# B&R Automation Studio project dbserv_0640 (part 5)

#### dbserv.c
```c
#ifdef _DEFAULT_INCLUDES
	#include <AsDefault.h>
#endif

/******************************************************************************
*    COPYRIGHT    BERNECKER + RAINER Industrie-Elektronik Ges.m.b.H           *
*******************************************************************************
*  Projekt:  DbServ
*  Teil:     Prozessabbild-Aufbau
*  Datei:    dbserv.c
*  Typ:      GNU-C (32 Bit)
*------------------------------------------------------------------------------
*  Revision: 01.03
*  Datum:    26-07-2004
*  Autor:    Martin Kurtz / MKrz
*------------------------------------------------------------------------------
*  Funktion: Task-Source-Datei.
*------------------------------------------------------------------------------
*  Rev.  | Datum    | Name | Kommentar
*  ------+----------+------+---------------------------------------------------
*  01.03 | 26-07-04 | MKrz | Nichtangabe von Item.Name für nicht verwendete Fubinstanzen
*        |          |      | führt zu keinen Logbucheinträgen;
*  01.02 | 15-07-04 | MKrz | Fehlerbeseitigung bei Logbuch-Fehlereintrag;
*  01.01 | 06-07-04 | MKrz | Fehlerbeseitigung Eventblockverwaltung;
*        |          |      | Parserfunktion für Timeout, Port, Client.Anz, App.Anz
*  01.00 | 04-08-03 | MKrz | Datei-Erstellung
*  02.00 | 10-07-26 | BIE  | strnicmp gegen strncasecmp ersetzt
*        |          |      |
******************************************************************************/

/***********************************************************************/
/* Headerfiles einbinden                                               */
/***********************************************************************/
#include <bur\plc.h>		/* RPS-spezifische Typendeklarationen */
#include <sys_lib.h>		/* System-Library */

#include <dataobj.h>
#include <fileio.h>
#include <brsystem.h>

#include <string.h>			/* String-Library */
#include <stdlib.h>			/* String-Library */

#include "platform.h"		/* CPU-Plattform */

#include "bksys.h"			/* Burklimat-Library */

#include "parser.h"			/* Parser-Library */
#include "dbserv.h"			/* BkTcp-Library */

#include <dbslib.h>

//unsigned short itoa(signed long value, unsigned long pString);

/***********************************************************************/
/* Variablendeklaration                                                */
/***********************************************************************/

/**** globale Variablen ************************************************/

/**** lokale Variablen *************************************************/

/* Anzahl Fehlerzaehler fuer ErrStatistics */
/*#define ERRCNTANZ				300*/

/* Struktur fuer Fehler-Statistik */
/*typedef struct {
	unsigned short	LastWarn;
	unsigned short	LastErr;
	unsigned short	Init;
	Timestamp_Typ	LastInit;
	unsigned short	ErrCount[ERRCNTANZ];
} Stats_Typ;*/

_LOCAL_RETAIN Stats_Typ		SYS_Statistic	;

_LOCAL_RETAIN	unsigned short	ParserState	;

_LOCAL_RETAIN	BIT				DbsTypeChanged, DbsPointChanged	;
		void  			*pDA_Data;
_LOCAL_RETAIN	UDINT			SizeDA_Data	;

_LOCAL	DatObjInfo_typ		iDatObjInfo;
_LOCAL	DatObjDelete_typ	iDatObjDelete;
_LOCAL	DatObjCreate_typ	iDatObjCreate;

_LOCAL_RETAIN	unsigned short	CountLines	;
_LOCAL_RETAIN	signed short	State_find_StationTypPoint, State_find_Section, State_find_Data	;
		short			StateGetDpInfo;

		unsigned char	*pParser, *pParserLine, *pParserErr;
		unsigned short	SectionType;
		unsigned char	*pDataArg1, *pDataArg2, *pDataArg3, *pTempStation, *pTempSection, *pTempPoint, *pTempData, *pDbsTypeFileBufferSize, *pDbsTypeFileBufferMode;
		unsigned short	SizeArg1, SizeArg2, SizeArg3 ;

_LOCAL	unsigned short	PortNumber, TimeoutValue;
_LOCAL	long			BufEvents, BufType;

		unsigned char	flagDbsUnit, flagDbsType, flagDbsPoint, flagDbsFub, flag, flagDbsExistPoints, flagDbsNotExistPoints, flagDbsFubInstance;
_LOCAL_RETAIN	unsigned short	maxDbsUnit, maxUsedUnit, DbsUnit, DbsType, maxDbsType, maxUsedType, DbsPoint, DbsItem	;
_LOCAL	unsigned char	DbsMemTypeData, DbsMemTypeEvent;
_LOCAL_RETAIN	unsigned long	memSize, SmemSize, StmpSize	;
		unsigned short	StateTMP_alloc;

_LOCAL_RETAIN	unsigned short	countStationTypPoint, countSection, countItem, countTimeItem	;
_LOCAL	unsigned short	countDefinedType, countDefinedPoint, countDefinedItem, countPortData, countTimeoutData, countEventData, countTypeData, countUnitData, countPointData	;
_LOCAL	unsigned short	countFub, countData, countExistPoints, countNotExistPoints, countNotDefinedItems, countInvalidExistItems, countNotExistItems, countLogMessages, countFubInstance	;
_LOCAL_RETAIN	unsigned short	countEventInstance, countWriteInstance	;

_LOCAL	unsigned short	SizeNameType, SizeNamePoint, SizeNameItem, sizeType, lenItem	;
_LOCAL_RETAIN	unsigned char	sItem, idTypeItem	;

		char			logBuffer[128];
		unsigned short	sMsgMaxLen;
_LOCAL_RETAIN	short			SwVersion	;

		unsigned short	i, j;
		unsigned char	DtIdx;
		unsigned short	DpIdx;

_LOCAL_RETAIN	unsigned char	go	;
_LOCAL_RETAIN	short			AnzWaitCycleDbs	;
		unsigned char	ErrStatisticsYField[EC_MAX / 8 + 1];

_LOCAL	TYPE_DESC		*pTypeDesc, *pWorkTypeDesc, *pInfoTypeDesc;
_LOCAL	ITEM_DESC		*pItemDesc, *pWorkItemDesc, *pInfoItemDesc;
_LOCAL	POINT_DESC		*pPointDesc, *pWorkPointDesc, *pInfoPointDesc;
_LOCAL	FUB_DESC		*pFubInstanceDesc;
_LOCAL_RETAIN	unsigned short	infoType, infoPoint	;
_LOCAL_RETAIN	unsigned char	*pTypeName, *pWorkTypeName, *pPointName, *pWorkPointName, *pWorkItemName, InfoTypeName[16], PointName[64]	;
		unsigned short	lenTypeName, lenPointName;
		unsigned long	len;

_LOCAL	ACCESS_SERVER		*idBrServer,	*pAccessServer;
		ACCESS_UNIT			*pAccessUnit;
		ACCESS_TYPE			*pAccessType,	*pAccessTypeWork;
		ACCESS_POINT		*pAccessPoint,	*pAccessPointWork;
		ACCESS_DATA			*pAccessData,	*pAccessDataWork;
		ACCESS_FUB_INSTANCE	*pAccessFubInstance;

		ACCESS_EVENT_PIPE	*pEventPipe;
		EVENT_PIPE_INSTANCE	*pEventPipeInstance;
		EVENT_PIPE_HEADER	*pEventPipeHeader;
		ACCESS_WRITE_PIPE	*pWritePipe;
		WRITE_PIPE_HEADER	*pWritePipeHeader;

_LOCAL_RETAIN	UINT			stateFubInstance	;
_LOCAL	UDINT			pFubInstance, lenFubInstance	;

/*_LOCAL	FUB_REF			x;*/

_LOCAL_RETAIN	USINT		bValue	;
_LOCAL_RETAIN	RTCtime_typ	RTCTime	;

_LOCAL	FileCreate_typ	iFileCreate;
_LOCAL	DevMemInfo_typ	iDevMemInfo;
_LOCAL	BOOL	filetest;
_LOCAL	USINT	buffer1[32], buffer2[32];

_LOCAL	SysInfo_typ		iSysInfo;

/***********************************************************************/
/* Initialisierungs-Unterprogramm                                      */
/***********************************************************************/

void _INIT init(void)
{
	idBrServer = NULL;
	SwVersion = BK_VERSION_NR;

	SYS_Statistic = SYS_Statistic;

	PortNumber = cTCP_DEFAULT_PORT;
	TimeoutValue = cTCP_DEFAULT_TIMEOUT;

	BufEvents = 0;
	BufType = 0;

	ParserState = cCD_PARSER_STATE_DEF_TCP;
	memset(ErrStatisticsYField, 0, sizeof(ErrStatisticsYField));

	AnzWaitCycleDbs = 0;

	countEventInstance = 8;
	countWriteInstance = 4;

	DbsTypeChanged = TRUE;
	DbsPointChanged = TRUE;

	go = TRUE;
}

/***********************************************************************/
/* zyklisches Hauptprogramm                                            */
/***********************************************************************/
void _CYCLIC cyclic(void)
{
	if (filetest == TRUE) {
		strcpy(buffer1, "Test");
		ultoa(i, buffer2);
		strcat(buffer1, buffer2);

		iFileCreate.enable = 1;
		iFileCreate.pDevice = (unsigned long)"CompactFlash";
		iFileCreate.pFile = (unsigned long)buffer1;
		FileCreate(&iFileCreate);
		if (iFileCreate.status == 0) {
			filetest = FALSE;
			i++;
		}
		else if (iFileCreate.status != 65535) {
			filetest = FALSE;
			i++;
		}
	}

	/* ----------------- */
	/* Start-Verzögerung */
	/* ----------------- */
	if (AnzWaitCycleDbs < ANZ_WAIT_CYCLE_TCP) {
		AnzWaitCycleDbs++;
		return;
	}

	/* ------------- */
	/* Parser - Lauf */
	/* ------------- */
	if (go == TRUE) {

		/* --- */
		/* DFA */
		/* --- */
		/*while (ParserState < cCD_PARSER_STATE_READY) {*/

			/* ------------- */
			/* DFA - Zustand */
			/* ------------- */
			switch (ParserState) {

				/* ============================= */
				/* DFA-Zustand: Tcp-Definitionen */
				/* ============================= */
				case cCD_PARSER_STATE_DEF_TCP:

					iDatObjInfo.enable = TRUE;
					iDatObjInfo.pName = (UDINT)cKW_DBS_DM_DP_LIST;
					DatObjInfo(&iDatObjInfo);
					if (iDatObjInfo.status == 0) {
						pDA_Data = (unsigned char*)iDatObjInfo.pDatObjMem;
						SizeDA_Data = iDatObjInfo.len;

						/* go */

						/* Datenmodul von Anfang an Parsen ... */
						CountLines = 0;
						pParser = (unsigned char*)pDA_Data;

						/* Zähler rücksetzen */
						countPortData = 0;
						countTimeoutData = 0;
						countStationTypPoint = 0;

						/* Parser-Status loeschen */
						State_find_StationTypPoint = 0;
						State_find_Section = 0;
						State_find_Data = 0;

						/* ------ */
						/* Parsen */
						/* ------ */
						while (pParser < (unsigned char*)pDA_Data + SizeDA_Data) {

							/* Suche nach Stations/Typ/Punkt-Beschreibung */
							State_find_StationTypPoint = find_StationTypPoint(pDA_Data, pParser, pDA_Data + SizeDA_Data,
																				&pParser, &pParserLine, &pParserErr, &CountLines,
																				&pDataArg1, &SizeArg1,
																				&pDataArg2, &SizeArg2,
																				&SectionType);
							/* keine Daten oder Fehler aufgetreten ? */
							if (State_find_StationTypPoint < 0) {
								break;
							}
							else {
								countStationTypPoint++;
							}

							/* Pointer auf Station/Typ/Punkt */
							switch (SectionType) {

								/* ------------------ */
								/* Stations-Abschnitt */
								/* ------------------ */
								case cCD_STATION:
									countSection = 0;
									do {
										State_find_Section = find_Section(pDA_Data, pParser, pDA_Data + SizeDA_Data,
																			&pParser, &pParserLine, &pParserErr, &CountLines,
																			&pDataArg1, &SizeArg1,
																			&pDataArg2, &SizeArg2,
																			cKW_TCP_SECTION);
										/* keine Daten oder Fehler aufgetreten ? */
										if (State_find_Section < 0) {
											break;
										}
										else {
											countSection++;
										}

										/* Pointer auf Anfang der Sektion stellen */
										if (pDataArg2 != NULL) {
											pParser = pDataArg2;
										}
										else {
											continue;
										}

										/* alle Daten der Sektion bearbeiten */
										countData = 0;
										do {
											/* Daten der Sektion anfordern */
											State_find_Data = find_Data(pDA_Data, pParser, pDA_Data + SizeDA_Data,
																		  &pParser, &pParserLine, &pParserErr, NULL,
																		  &pDataArg1, &SizeArg1,
																		  &pDataArg2, &SizeArg2,
																		  &pDataArg3, &SizeArg3);
											/* keine Daten oder Fehler aufgetreten ? */
											if (State_find_Data < -1) {
												break;
											}
											else if (State_find_Data == -1) {
												if (pParser < (unsigned char*)pDA_Data + SizeDA_Data) {
													pParser++;
													State_find_Data = TRUE;
													continue;
												}
												else {
													break;
												}
											}
											else {
												/* Port-Bezeichner */
												if (strlen(cKW_TCP_PORT) == SizeArg1 && strncasecmp(pDataArg1, cKW_TCP_PORT, SizeArg1) == 0 &&
													strlen(cKW_TCP_PORT_NUMBER) == SizeArg2 && strncasecmp(pDataArg2, cKW_TCP_PORT_NUMBER, SizeArg2) == 0 &&
													pDataArg3 != NULL && SizeArg3 != 0 &&
													IsANumber(pDataArg3) == TRUE)
												{
													countPortData++;
													PortNumber = atoi(pDataArg3);
												}
												/* Timeout-Bezeichner */
												else if (strlen(cKW_TCP_TIMEOUT) == SizeArg1 && strncasecmp(pDataArg1, cKW_TCP_TIMEOUT, SizeArg1) == 0 &&
													strlen(cKW_TCP_TIMEOUT_NUMBER) == SizeArg2 && strncasecmp(pDataArg2, cKW_TCP_TIMEOUT_NUMBER, SizeArg2) == 0 &&
													pDataArg3 != NULL && SizeArg3 != 0 &&
													IsANumber(pDataArg3) == TRUE)
												{
													countTimeoutData++;
													TimeoutValue = atoi(pDataArg3);
												}
												/* unbekannte Zuweisung */
												else {
												}
											}
										} while (State_find_Data == TRUE);
									} while (State_find_Section == TRUE);
									break;
							} /* (SectionType) */
						} /* (pParser < (unsigned char*)pDA_Data + SizeDA_Data) */

						/* ---------------- */
						/* nächster Zustand */
						/* ---------------- */
						ParserState = cCD_PARSER_STATE_DEF_BUF;

					} /* (DA_DataOk == TRUE) */
					else {
						/* Fehler beim Datenmodul */
						ErrStatistics("dbserv", ERRLOG, EC_DA_NOT_FOUND + EC_DBS_BASE, CountLines, ERR_DBS_PRE, ET_DA_NOT_FOUND);
						ParserState = cCD_PARSER_STATE_ERROR;
					}
					break;

				/* ============================= */
				/* DFA-Zustand: Buf-Definitionen */
				/* ============================= */
				case cCD_PARSER_STATE_DEF_BUF:

					iDatObjInfo.enable = TRUE;
					iDatObjInfo.pName = (UDINT)cKW_DBS_DM_DP_LIST;
					DatObjInfo(&iDatObjInfo);
					if (iDatObjInfo.status == 0) {
						pDA_Data = (unsigned char*)iDatObjInfo.pDatObjMem;
						SizeDA_Data = iDatObjInfo.len;

						/* go */

						/* Datenmodul von Anfang an Parsen ... */
						CountLines = 0;
						pParser = (unsigned char*)pDA_Data;

						/* Zähler rücksetzen */
						countEventData = 0;
						countTypeData = 0;
						countStationTypPoint = 0;

						/* Parser-Status loeschen */
						State_find_StationTypPoint = 0;
						State_find_Section = 0;
						State_find_Data = 0;

						/* ------ */
						/* Parsen */
						/* ------ */
						while (pParser < (unsigned char*)pDA_Data + SizeDA_Data) {

							/* Suche nach Stations/Typ/Punkt-Beschreibung */
							State_find_StationTypPoint = find_StationTypPoint(pDA_Data, pParser, pDA_Data + SizeDA_Data,
																				&pParser, &pParserLine, &pParserErr, &CountLines,
																				&pDataArg1, &SizeArg1,
																				&pDataArg2, &SizeArg2,
																				&SectionType);
							/* keine Daten oder Fehler aufgetreten ? */
							if (State_find_StationTypPoint < 0) {
								break;
							}
							else {
								countStationTypPoint++;
							}

							/* Pointer auf Station/Typ/Punkt */
							switch (SectionType) {

								/* ------------------ */
								/* Stations-Abschnitt */
								/* ------------------ */
								case cCD_STATION:
									countSection = 0;
									do {
										State_find_Section = find_Section(pDA_Data, pParser, pDA_Data + SizeDA_Data,
																			&pParser, &pParserLine, &pParserErr, &CountLines,
																			&pDataArg1, &SizeArg1,
																			&pDataArg2, &SizeArg2,
																			cKW_BUF_SECTION);
										/* keine Daten oder Fehler aufgetreten ? */
										if (State_find_Section < 0) {
											break;
										}
										else {
											countSection++;
										}

										/* Pointer auf Anfang der Sektion stellen */
										if (pDataArg2 != NULL) {
											pParser = pDataArg2;
										}
										else {
											continue;
										}

										/* alle Daten der Sektion bearbeiten */
										countData = 0;
										do {
											/* Daten der Sektion anfordern */
											State_find_Data = find_Data(pDA_Data, pParser, pDA_Data + SizeDA_Data,
																		  &pParser, &pParserLine, &pParserErr, NULL,
																		  &pDataArg1, &SizeArg1,
																		  &pDataArg2, &SizeArg2,
																		  &pDataArg3, &SizeArg3);
											/* keine Daten oder Fehler aufgetreten ? */
											if (State_find_Data < -1) {
												break;
											}
											else if (State_find_Data == -1) {
												if (pParser < (unsigned char*)pDA_Data + SizeDA_Data) {
													pParser++;
													State_find_Data = TRUE;
													continue;
												}
												else {
													break;
												}
											}
											else {
												/* Events-Bezeichner */
												if (strlen(cKW_DBS_BUF_EVENTS) == SizeArg1 && strncasecmp(pDataArg1, cKW_DBS_BUF_EVENTS, SizeArg1) == 0 &&
													pDataArg2 == NULL &&
													pDataArg3 != NULL && SizeArg3 != 0 &&
													IsANumber(pDataArg3) == TRUE)
												{
													countEventData++;
													BufEvents = atoi(pDataArg3);
												}
												/* Typ-Bezeichner */
												else if (strlen(cKW_DBS_BUF_TYPE) == SizeArg2 && strncasecmp(pDataArg2, cKW_DBS_BUF_TYPE, SizeArg2) == 0 &&
													pDataArg2 == NULL &&
													pDataArg3 != NULL && SizeArg3 != 0 &&
													IsANumber(pDataArg3) == TRUE)
												{
													countTypeData++;
													BufType = atoi(pDataArg3);
												}
												/* unbekannte Zuweisung */
												else {
												}
											}
										} while (State_find_Data == TRUE);
									} while (State_find_Section == TRUE);
									break;
							} /* (SectionType) */
						} /* (pParser < (unsigned char*)pDA_Data + SizeDA_Data) */

						/* ---------------- */
						/* nächster Zustand */
						/* ---------------- */
						ParserState = cCD_PARSER_STATE_COUNT_TYPE;

					} /* (DA_DataOk == TRUE) */
					else {
						/* Fehler beim Datenmodul */
						ErrStatistics("dbserv", ERRLOG, EC_DA_NOT_FOUND + EC_DBS_BASE, CountLines, ERR_DBS_PRE, ET_DA_NOT_FOUND);
						ParserState = cCD_PARSER_STATE_ERROR;
					}
					break;

				/* ====================================== */
				/* DFA-Zustand: Zählen der DBS-Datentypen */
				/* ====================================== */
				case cCD_PARSER_STATE_COUNT_TYPE:

					idBrServer = NULL;

					iDatObjInfo.enable = TRUE;
					iDatObjInfo.pName = (UDINT)cKW_DBS_DM_TYP_LIST;
					DatObjInfo(&iDatObjInfo);
					if (iDatObjInfo.status == 0) {
						pDA_Data = (unsigned char*)iDatObjInfo.pDatObjMem;
						SizeDA_Data = iDatObjInfo.len;

						SmemSize = 0, StmpSize = 0;

						/* go */

						/* Datenmodul von Anfang an Parsen ... */
						CountLines = 0;
						pParser = (unsigned char*)pDA_Data;

						/* Zähler rücksetzen */
						countDefinedType = 0;
						countDefinedItem = 0;
						countPortData = 0;
						countTimeoutData = 0;
						countExistPoints = 0;
						countNotExistPoints = 0;
						countStationTypPoint = 0;
						countLogMessages = 0;

						SizeNameType = 0, SizeNameItem = 0;

						/* Parser-Status loeschen */
						State_find_StationTypPoint = 0;
						State_find_Section = 0;
						State_find_Data = 0;

						/* ------ */
						/* Parsen */
						/* ------ */
						while (pParser < (unsigned char*)pDA_Data + SizeDA_Data) {

							/* Suche nach Stations/Typ/Punkt-Beschreibung */
							State_find_StationTypPoint = find_StationTypPoint(pDA_Data, pParser, pDA_Data + SizeDA_Data,
																				&pParser, &pParserLine, &pParserErr, &CountLines,
																				&pDataArg1, &SizeArg1,
																				&pDataArg2, &SizeArg2,
																				&SectionType);
							/* keine Daten oder Fehler aufgetreten ? */
							if (State_find_StationTypPoint < 0) {
								break;
							}
							else {
								countStationTypPoint++;
							}

							/* Pointer auf Station/Typ/Punkt */
							switch (SectionType) {

								/* ------------- */
								/* Typ-Abschnitt */
								/* ------------- */
								case cCD_TYP:

									countDefinedType++;
									SizeNameType += SizeArg1 + 1;
									countItem = 0, sizeType = 0;
									countSection = 0;
									do {
										State_find_Section = find_Section(pDA_Data, pParser, pDA_Data + SizeDA_Data,
																			&pParser, &pParserLine, &pParserErr, &CountLines,
																			&pDataArg1, &SizeArg1,
																			&pDataArg2, &SizeArg2,
																			cKW_ALL_SECTION);
										/* keine Daten oder Fehler aufgetreten ? */
										if (State_find_Section < 0) {
											break;
										}
										else {
											countSection++;
										}

										/* Pointer auf Anfang der Sektion stellen */
										if (pDataArg2 != NULL) {
											pParser = pDataArg2;
										}
										else {
											continue;
										}

										/* alle Daten der Sektion bearbeiten */
										countData = 0;
										do {
											/* Daten der Sektion anfordern */
											State_find_Data = find_Data(pDA_Data, pParser, pDA_Data + SizeDA_Data,
																		  &pParser, &pParserLine, &pParserErr, NULL,
																		  &pDataArg1, &SizeArg1,
																		  &pDataArg2, &SizeArg2,
																		  &pDataArg3, &SizeArg3);
											/* keine Daten oder Fehler aufgetreten ? */
											if (State_find_Data < 0) {
												break;
											}
											else {
												/* Typ-Bezeichner */
												if (strlen(cKW_DBS_TYPE) == SizeArg1 && strncasecmp(pDataArg1, cKW_DBS_TYPE, SizeArg1) == 0 &&
													strlen(cKW_DBS_TYPE_NUMBER) == SizeArg2 && strncasecmp(pDataArg2, cKW_DBS_TYPE_NUMBER, SizeArg2) == 0 &&
													pDataArg3 != NULL && SizeArg3 != 0 &&
													IsANumber(pDataArg3) == TRUE)
												{
													if (atoi(pDataArg3) >= 0 && atoi(pDataArg3) <= cMAX_TYPE_DEF) {
														DbsType = atoi(pDataArg3);
														maxDbsType = (maxDbsType > DbsType) ? maxDbsType : DbsType;
													}
													else {
													}
												}
											}
										} while (State_find_Data == TRUE);
									} while (State_find_Section == TRUE);
									break;

								/* -------------- */
								/* Item-Abschnitt */
								/* -------------- */
								case cCD_ITEM:

									do {
										State_find_Section = find_Section(pDA_Data, pParser, pDA_Data + SizeDA_Data,
																			&pParser, &pParserLine, &pParserErr, &CountLines,
																			&pDataArg1, &SizeArg1,
																			&pDataArg2, &SizeArg2,
																			cKW_ALL_SECTION);
										/* keine Daten oder Fehler aufgetreten ? */
										if (State_find_Section < 0) {
											break;
										}
										else {
											countItem++;
										}

										/* Pointer auf Anfang der Sektion stellen */
										if (pDataArg2 != NULL) {
											pParser = pDataArg2;
										}
										else {
											continue;
										}

										/* alle Daten der Sektion bearbeiten */
										countData = 0;
										do {
											/* Daten der Sektion anfordern */
											State_find_Data = find_Data(pDA_Data, pParser, pDA_Data + SizeDA_Data,
																		  &pParser, &pParserLine, &pParserErr, NULL,
																		  &pDataArg1, &SizeArg1,
																		  &pDataArg2, &SizeArg2,
																		  &pDataArg3, &SizeArg3);
											/* keine Daten oder Fehler aufgetreten ? */
											if (State_find_Data < 0) {
												break;
											}
											else {
												/* Typ-Bezeichner */
												if (strlen(cKW_DBS_TYPE) == SizeArg1 && strncasecmp(pDataArg1, cKW_DBS_TYPE, SizeArg1) == 0) {
													/* BOOL */
													if (strlen(cKW_DBS_TYPE_BOOL) == SizeArg3 && strncmp(pDataArg3, cKW_DBS_TYPE_BOOL, SizeArg3) == 0) {
														countDefinedItem++;
														sizeType += sizeof(BOOL);
													}
													/* USINT */
													else if (strlen(cKW_DBS_TYPE_USINT) == SizeArg3 && strncmp(pDataArg3, cKW_DBS_TYPE_USINT, SizeArg3) == 0) {
														countDefinedItem++;
														sizeType += sizeof(USINT);
													}
													/* SINT */
													else if (strlen(cKW_DBS_TYPE_SINT) == SizeArg3 && strncmp(pDataArg3, cKW_DBS_TYPE_SINT, SizeArg3) == 0) {
														countDefinedItem++;
														sizeType += sizeof(SINT);
													}
													/* UINT */
													else if (strlen(cKW_DBS_TYPE_UINT) == SizeArg3 && strncmp(pDataArg3, cKW_DBS_TYPE_UINT, SizeArg3) == 0) {
														countDefinedItem++;
														sizeType += sizeof(UINT);
													}
													/* INT */
													else if (strlen(cKW_DBS_TYPE_INT) == SizeArg3 && strncmp(pDataArg3, cKW_DBS_TYPE_INT, SizeArg3) == 0) {
														countDefinedItem++;
														sizeType += sizeof(INT);
													}
													/* UDINT */
													else if (strlen(cKW_DBS_TYPE_UDINT) == SizeArg3 && strncmp(pDataArg3, cKW_DBS_TYPE_UDINT, SizeArg3) == 0) {
														countDefinedItem++;
														sizeType += sizeof(UDINT);
													}
													/* DINT */
													else if (strlen(cKW_DBS_TYPE_DINT) == SizeArg3 && strncmp(pDataArg3, cKW_DBS_TYPE_DINT, SizeArg3) == 0) {
														countDefinedItem++;
														sizeType += sizeof(DINT);
													}
													/* STREAM */
													else if (strlen(cKW_DBS_TYPE_STREAM) == SizeArg3 && strncmp(pDataArg3, cKW_DBS_TYPE_STREAM, SizeArg3) == 0) {
														countDefinedItem++;
														sizeType += 2 * sizeof(UDINT);
													}
													/* sonst */
													else {
														continue;
													}
												}
												/* Zeitstempel-Bezeichner */
												else if (strlen(cKW_DBS_TYPE_TIMESTAMP) == SizeArg1 && strncasecmp(pDataArg1, cKW_DBS_TYPE_TIMESTAMP, SizeArg1) == 0 &&
													pDataArg3 != NULL && SizeArg3 != 0 &&
													IsANumber(pDataArg3) == TRUE)
												{
												}
												/* Item-Bezeichner */
												else if (strlen(cKW_DBS_ITEM) == SizeArg1 && strncasecmp(pDataArg1, cKW_DBS_ITEM, SizeArg1) == 0 &&
													strlen(cKW_DBS_ITEM_NAME) == SizeArg2 && strncasecmp(pDataArg2, cKW_DBS_ITEM_NAME, SizeArg2) == 0 &&
													pDataArg3 != NULL && SizeArg3 != 0)
												{
													SizeNameItem += SizeArg3 + 1;
												}
											}
										} while (State_find_Data == TRUE);
									} while (State_find_Section == TRUE);
									break;

							} /* (SectionType) */
						} /* (pParser < (unsigned char*)pDA_Data + SizeDA_Data) */

						/* ---------------- */
						/* nächster Zustand */
						/* ---------------- */
						ParserState = cCD_PARSER_STATE_DEF_TYPE;

					} /* (DA_DataOk == TRUE) */
					else {
						/* Fehler beim Datenmodul */
						ErrStatistics("dbserv", ERRLOG, EC_DA_NOT_FOUND + EC_DBS_BASE, CountLines, ERR_DBS_PRE, ET_DA_NOT_FOUND);
						ParserState = cCD_PARSER_STATE_ERROR;
					}
					break;

				/* ==================================================================== */
				/* DFA-Zustand: Speicher allokieren und Aufbau der Bäume für Datentypen */
				/* ==================================================================== */
				case cCD_PARSER_STATE_DEF_TYPE:
					memSize = (maxDbsType + 1) * sizeof(TYPE_DESC)
							+ countDefinedItem * sizeof(ITEM_DESC)
							+ SizeNameType
							+ SizeNameItem;
					if (memSize > 0) {
						StateTMP_alloc = TMP_alloc(memSize, (void*)&pTypeDesc);
						if (StateTMP_alloc == 0) {
							SmemSize += 0;
							StmpSize += memSize;
							memset(pTypeDesc, 0, memSize);

							/* initialisieren */
							for (i=0; i<=maxDbsType; i++) {
								pTypeDesc[i].dbsType--;
							}

							pItemDesc = (ITEM_DESC*)(pTypeDesc + (maxDbsType + 1));
							pWorkItemDesc = pItemDesc;
							pWorkTypeName = (unsigned char*)(pItemDesc + countDefinedItem);
							pWorkItemName = pWorkTypeName + SizeNameType;

							/* Datenmodul von Anfang an Parsen ... */
							CountLines = 0;
							pParser = (unsigned char*)pDA_Data;

							/* Zähler rücksetzen */
							countDefinedType = 0;
							countDefinedItem = 0;
							countPortData = 0;
							countTimeoutData = 0;
							countExistPoints = 0;
							countNotExistPoints = 0;
							countStationTypPoint = 0;
							countLogMessages = 0;

							SizeNameType = 0;

							/* Parser-Status loeschen */
							State_find_StationTypPoint = 0;
							State_find_Section = 0;
							State_find_Data = 0;

							/* ------ */
							/* Parsen */
							/* ------ */
							while (pParser < (unsigned char*)pDA_Data + SizeDA_Data) {

								/* Suche nach Stations/Typ/Punkt-Beschreibung */
								State_find_StationTypPoint = find_StationTypPoint(pDA_Data, pParser, pDA_Data + SizeDA_Data,
																					&pParser, &pParserLine, &pParserErr, &CountLines,
																					&pDataArg1, &SizeArg1,
																					&pDataArg2, &SizeArg2,
																					&SectionType);
								/* keine Daten oder Fehler aufgetreten ? */
								if (State_find_StationTypPoint < 0) {
									break;
								}
								else {
									countStationTypPoint++;
								}

								/* Pointer auf Station/Typ/Punkt */
								switch (SectionType) {

									/* ------------- */
									/* Typ-Abschnitt */
									/* ------------- */
									case cCD_TYP:

										countDefinedType++;
										SizeNameType += SizeArg1 + 1;
										pTypeName = pDataArg1, lenTypeName = SizeArg1;
										DbsItem = 0;
										countItem = 0, sizeType = 0;
										countSection = 0;

										pDbsTypeFileBufferSize = NULL, pDbsTypeFileBufferMode = NULL;

										do {
											State_find_Section = find_Section(pDA_Data, pParser, pDA_Data + SizeDA_Data,
																				&pParser, &pParserLine, &pParserErr, &CountLines,
																				&pDataArg1, &SizeArg1,
																				&pDataArg2, &SizeArg2,
																				cKW_ALL_SECTION);
											/* keine Daten oder Fehler aufgetreten ? */
											if (State_find_Section < 0) {
												break;
											}
											else {
												countSection++;
											}

											/* Pointer auf Anfang der Sektion stellen */
											if (pDataArg2 != NULL) {
												pParser = pDataArg2;
											}
											else {
												continue;
											}

											/* alle Daten der Sektion bearbeiten */
											countData = 0;
											do {
												/* Daten der Sektion anfordern */
												State_find_Data = find_Data(pDA_Data, pParser, pDA_Data + SizeDA_Data,
																			  &pParser, &pParserLine, &pParserErr, NULL,
																			  &pDataArg1, &SizeArg1,
																			  &pDataArg2, &SizeArg2,
																			  &pDataArg3, &SizeArg3);
												/* keine Daten oder Fehler aufgetreten ? */
												if (State_find_Data < 0) {
													break;
												}
												else {
													/* Typ-Bezeichner */
													if (strncasecmp(pDataArg1, cKW_DBS_TYPE, SizeArg1) == 0 && strlen(cKW_DBS_TYPE) == SizeArg1 &&
														strncasecmp(pDataArg2, cKW_DBS_TYPE_NUMBER, SizeArg2) == 0 && strlen(cKW_DBS_TYPE_NUMBER) == SizeArg2 &&
														pDataArg3 != NULL && SizeArg3 != 0 &&
														IsANumber(pDataArg3) == TRUE)
													{
														DbsType = atoi(pDataArg3);
														/* Typnummer bereits vergeben ? */
														if (pTypeDesc[DbsType].dbsType != DbsType) {
															pTypeDesc[DbsType].dbsType = DbsType;
															/* Typname bereits vergeben ? */
															flag = FALSE;
															for (i=0; i<=maxDbsType; i++) {
																if (pTypeDesc[i].pTypeName != NULL) {
																	if (strlen(pTypeDesc[i].pTypeName) == lenTypeName &&
																		strncmp(pTypeDesc[i].pTypeName, pTypeName, strlen(pTypeDesc[i].pTypeName)) == 0)
																	{
																		flag = TRUE;
																		break;
																	}
																}
															}
															if (flag == FALSE) {
																if (pTypeDesc[DbsType].pTypeName == NULL) {
																	pTypeDesc[DbsType].pTypeName = pWorkTypeName;
																}
																strncpy(pTypeDesc[DbsType].pTypeName, pTypeName, lenTypeName);
																pWorkTypeName = pWorkTypeName + lenTypeName + 1;
															}
															else {
																strcat(strcat(strcpy(logBuffer, (char*)iDatObjInfo.pName), ET_TYPE_ALREADY_EXIST), "\n");
																strcat(strncat(logBuffer, pTypeName, lenTypeName), "\n");
																strncat(logBuffer, pDataArg1, pDataArg3 - pDataArg1 + SizeArg3);
																ErrStatistics("dbserv", ERRLOG, EC_TYPE_ALREADY_EXIST + EC_DBS_BASE, CountLines, ERR_DBS_PRE, logBuffer);
															}
														} /* (pTypeDesc[DbsType].dbsType != DbsType) */
														else {
															/* !!! CHECK !!! */
															strcat(strcat(strcpy(logBuffer, (char*)iDatObjInfo.pName), ET_TYPE_NO_INVALID), "\n");
															strcat(strncat(logBuffer, pTypeName, lenTypeName), "\n");
															strncat(logBuffer, pDataArg1, pDataArg3 - pDataArg1 + SizeArg3);
															ErrStatistics("dbserv", ERRLOG, EC_TYPE_NO_INVALID + EC_DBS_BASE, CountLines, ERR_DBS_PRE, logBuffer);
														}
													}
													/* FileBuffer Grösse */
													else if (strncasecmp(pDataArg1, cKW_DBS_TYPE, SizeArg1) == 0 && strlen(cKW_DBS_TYPE) == SizeArg1 &&
														strncasecmp(pDataArg2, cKW_DBS_TYPE_FILE_SIZE, SizeArg2) == 0 && strlen(cKW_DBS_TYPE_FILE_SIZE) == SizeArg2 &&
														pDataArg3 != NULL && SizeArg3 != 0 &&
														IsANumber(pDataArg3) == TRUE)
													{
														unsigned long	DbsTypeFileBufferSize;
														pDbsTypeFileBufferSize = pDataArg3;

														DbsTypeFileBufferSize = atoi(pDataArg3);
														pTypeDesc[DbsType].SizeFileBuffer = DbsTypeFileBufferSize;
														pTypeDesc[DbsType].FileBuffer = TRUE;
													}
													/* FileBuffer Modus */
													else if (strncasecmp(pDataArg1, cKW_DBS_TYPE, SizeArg1) == 0 && strlen(cKW_DBS_TYPE) == SizeArg1 &&
														strncasecmp(pDataArg2, cKW_DBS_TYPE_FILE_MODE, SizeArg2) == 0 && strlen(cKW_DBS_TYPE_FILE_MODE) == SizeArg2 &&
														pDataArg3 != NULL && SizeArg3 != 0 &&
														IsANumber(pDataArg3) == TRUE)
													{
														unsigned char	DbsTypeFileBufferMode;
														pDbsTypeFileBufferMode = pDataArg3;

														DbsTypeFileBufferMode = atoi(pDataArg3);
														pTypeDesc[DbsType].ModeFileBuffer = DbsTypeFileBufferMode;
													}

													/* Buf-Bezeichner */
													else if (strlen(cKW_DBS_BUF_ATTRIBUTE) == SizeArg1 && strncasecmp(pDataArg1, cKW_DBS_BUF_ATTRIBUTE, SizeArg1) == 0 &&
														pDataArg3 != NULL && SizeArg3 != 0 &&
														IsANumber(pDataArg3) == TRUE)
													{
														pTypeDesc[DbsType].FileBuffer = atoi(pDataArg3);
													}

												}
											} while (State_find_Data == TRUE);
										} while (State_find_Section == TRUE);

										/* FileBuffer Grösse */
										if (pDbsTypeFileBufferSize != NULL) {
											pTypeDesc[DbsType].SizeFileBuffer = atoi(pDbsTypeFileBufferSize);
											pTypeDesc[DbsType].FileBuffer = TRUE;
										}
										/* FileBuffer Modus */
										if (pDbsTypeFileBufferMode != NULL) {
											pTypeDesc[DbsType].ModeFileBuffer = atoi(pDbsTypeFileBufferMode);
										}
										break;

									/* -------------- */
									/* Item-Abschnitt */
									/* -------------- */
									case cCD_ITEM:

										do {
											State_find_Section = find_Section(pDA_Data, pParser, pDA_Data + SizeDA_Data,
																				&pParser, &pParserLine, &pParserErr, &CountLines,
																				&pDataArg1, &SizeArg1,
																				&pDataArg2, &SizeArg2,
																				cKW_ALL_SECTION);
											/* keine Daten oder Fehler aufgetreten ? */
											if (State_find_Section < 0) {
												break;
											}
											else {
												countItem++;
											}

											/* Pointer auf Anfang der Sektion stellen */
											if (pDataArg2 != NULL) {
												pParser = pDataArg2;
											}
											else {
												continue;
											}

											/* alle Daten der Sektion bearbeiten */
											countData = 0;
											do {
												/* Daten der Sektion anfordern */
												State_find_Data = find_Data(pDA_Data, pParser, pDA_Data + SizeDA_Data,
																			  &pParser, &pParserLine, &pParserErr, NULL,
																			  &pDataArg1, &SizeArg1,
																			  &pDataArg2, &SizeArg2,
																			  &pDataArg3, &SizeArg3);
												/* keine Daten oder Fehler aufgetreten ? */
												if (State_find_Data < 0) {
													break;
												}
												else {
													/* Typ-Bezeichner */
													if (strlen(cKW_DBS_TYPE) == SizeArg1 && strncasecmp(pDataArg1, cKW_DBS_TYPE, SizeArg1) == 0) {
														/* BOOL */
														if (strlen(cKW_DBS_TYPE_BOOL) == SizeArg3 && strncmp(pDataArg3, cKW_DBS_TYPE_BOOL, SizeArg3) == 0) {
															lenItem = sizeof(BOOL);
															sItem = FALSE;
															idTypeItem = cDBS_IDTYPE_BOOL;
														}
														/* USINT */
														else if (strlen(cKW_DBS_TYPE_USINT) == SizeArg3 && strncmp(pDataArg3, cKW_DBS_TYPE_USINT, SizeArg3) == 0) {
															lenItem = sizeof(USINT);
															sItem = FALSE;
															idTypeItem = cDBS_IDTYPE_USINT;
														}
														/* SINT */
														else if (strlen(cKW_DBS_TYPE_SINT) == SizeArg3 && strncmp(pDataArg3, cKW_DBS_TYPE_SINT, SizeArg3) == 0) {
															lenItem = sizeof(SINT);
															sItem = TRUE;
															idTypeItem = cDBS_IDTYPE_SINT;
														}
														/* UINT */
														else if (strlen(cKW_DBS_TYPE_UINT) == SizeArg3 && strncmp(pDataArg3, cKW_DBS_TYPE_UINT, SizeArg3) == 0) {
															lenItem = sizeof(UINT);
															sItem = FALSE;
															idTypeItem = cDBS_IDTYPE_UINT;
														}
														/* INT */
														else if (strlen(cKW_DBS_TYPE_INT) == SizeArg3 && strncmp(pDataArg3, cKW_DBS_TYPE_INT, SizeArg3) == 0) {
															lenItem = sizeof(INT);
															sItem = TRUE;
															idTypeItem = cDBS_IDTYPE_INT;
														}
														/* UDINT */
														else if (strlen(cKW_DBS_TYPE_UDINT) == SizeArg3 && strncmp(pDataArg3, cKW_DBS_TYPE_UDINT, SizeArg3) == 0) {
															lenItem = sizeof(UDINT);
															sItem = FALSE;
															idTypeItem = cDBS_IDTYPE_UDINT;
														}
														/* DINT */
														else if (strlen(cKW_DBS_TYPE_DINT) == SizeArg3 && strncmp(pDataArg3, cKW_DBS_TYPE_DINT, SizeArg3) == 0) {
															lenItem = sizeof(DINT);
															sItem = TRUE;
															idTypeItem = cDBS_IDTYPE_DINT;
														}
														/* STREAM */
														else if (strlen(cKW_DBS_TYPE_STREAM) == SizeArg3 && strncmp(pDataArg3, cKW_DBS_TYPE_STREAM, SizeArg3) == 0) {
															lenItem = 2 * sizeof(UDINT);
															sItem = TRUE;
															idTypeItem = cDBS_IDTYPE_STREAM;
														}
														/* sonst */
														else {
															continue;
														}
														/* Informationen in den Typdescriptor eintragen */
														if (pTypeDesc[DbsType].pItemDesc == NULL) {
															pTypeDesc[DbsType].pItemDesc = pWorkItemDesc;
														}
														pTypeDesc[DbsType].pItemDesc[DbsItem].offItem = sizeType;
														pTypeDesc[DbsType].pItemDesc[DbsItem].lenItem = lenItem;
														pTypeDesc[DbsType].pItemDesc[DbsItem].sItem = sItem;
														pTypeDesc[DbsType].pItemDesc[DbsItem].idTypeItem = idTypeItem;
														sizeType += lenItem;
													}
													/* Zeitstempel-Bezeichner */
													else if (strlen(cKW_DBS_TYPE_TIMESTAMP) == SizeArg1 && strncasecmp(pDataArg1, cKW_DBS_TYPE_TIMESTAMP, SizeArg1) == 0 &&
														pDataArg3 != NULL && SizeArg3 != 0 &&
														IsANumber(pDataArg3) == TRUE)
													{
														pTypeDesc[DbsType].pItemDesc[DbsItem].tsItem = atoi(pDataArg3);
													}

													/* Buf-Bezeichner */
													else if (strlen(cKW_DBS_BUF_ATTRIBUTE) == SizeArg1 && strncasecmp(pDataArg1, cKW_DBS_BUF_ATTRIBUTE, SizeArg1) == 0 &&
														pDataArg3 != NULL && SizeArg3 != 0 &&
														IsANumber(pDataArg3) == TRUE)
													{
														pTypeDesc[DbsType].FileBuffer = atoi(pDataArg3);
														pTypeDesc[DbsType].pItemDesc[DbsItem].FileBuffer = atoi(pDataArg3);
													}

													/* Item-Nummer */
													else if (strlen(cKW_DBS_ITEM) == SizeArg1 && strncasecmp(pDataArg1, cKW_DBS_ITEM, SizeArg1) == 0 &&
														strlen(cKW_DBS_ITEM_NUMBER) == SizeArg2 && strncasecmp(pDataArg2, cKW_DBS_ITEM_NUMBER, SizeArg2) == 0 &&
														pDataArg3 != NULL && SizeArg3 != 0 &&
														IsANumber(pDataArg3) == TRUE)
													{
														/* Itemnummer richtig ? */
														if (atoi(pDataArg3) + 1 != countItem) {
															/* !!! CHECK !!! */
															strcat(strcat(strcpy(logBuffer, (char*)iDatObjInfo.pName), ET_ITEM_NO_INVALID), "\n");
															strcat(strncat(logBuffer, pTypeName, lenTypeName), "\n");
															strncat(logBuffer, pDataArg1, pDataArg3 - pDataArg1 + SizeArg3);
															ErrStatistics("dbserv", ERRLOG, EC_ITEM_NO_INVALID + EC_DBS_BASE, CountLines, ERR_DBS_PRE, logBuffer);
														}
													}
													/* Item-Bezeichner */
													else if (strlen(cKW_DBS_ITEM) == SizeArg1 && strncasecmp(pDataArg1, cKW_DBS_ITEM, SizeArg1) == 0 &&
														strlen(cKW_DBS_ITEM_NAME) == SizeArg2 && strncasecmp(pDataArg2, cKW_DBS_ITEM_NAME, SizeArg2) == 0 &&
														pDataArg3 != NULL && SizeArg3 != 0)
													{
														/* Itemname bereits vergeben ? */
														flag = FALSE;
														for (i=0; i<countItem; i++) {
															if (pTypeDesc[DbsType].pItemDesc[i].pNameItem != NULL) {
																if (strlen(pTypeDesc[DbsType].pItemDesc[i].pNameItem) == SizeArg3 &&
																	strncmp(pTypeDesc[DbsType].pItemDesc[i].pNameItem, pDataArg3, SizeArg3) == 0) {
																	flag = TRUE;
																	break;
																}
															}
														}
														if (flag == FALSE) {
															if (pTypeDesc[DbsType].pItemDesc[DbsItem].pNameItem == NULL) {
																pTypeDesc[DbsType].pItemDesc[DbsItem].pNameItem = pWorkItemName;
															}
															strncpy(pTypeDesc[DbsType].pItemDesc[DbsItem].pNameItem, pDataArg3, SizeArg3);
															pWorkItemName = pWorkItemName + SizeArg3 + 1;
														}
														else {
															pWorkItemName = pWorkItemName + 1;
															/* !!! CHECK !!! */
															strcat(strcat(strcpy(logBuffer, (char*)iDatObjInfo.pName), ET_ITEM_ALREADY_EXIST), "\n");
															strcat(strncat(logBuffer, pTypeName, lenTypeName), "\n");
															strncat(logBuffer, pDataArg1, pDataArg3 - pDataArg1 + SizeArg3);
															ErrStatistics("dbserv", ERRLOG, EC_ITEM_ALREADY_EXIST + EC_DBS_BASE, CountLines, ERR_DBS_PRE, logBuffer);
														}
													}
												}
											} while (State_find_Data == TRUE);
										} while (State_find_Section == TRUE);

										/* Informationen in den Typdescriptor eintragen */
										pTypeDesc[DbsType].sizeType = sizeType;
										pTypeDesc[DbsType].countItem = countItem;
										DbsItem++;
										pWorkItemDesc++;
										break;

								} /* (SectionType) */
							} /* (pParser < (unsigned char*)pDA_Data + SizeDA_Data) */

							/* ---------------- */
							/* nächster Zustand */
							/* ---------------- */
							ParserState = cCD_PARSER_STATE_COMPARE_DO_TYPE;

						} /* (StateTMP_alloc == 0) */
						else {
							/* Fehler bei StateTMP_alloc */
							ParserState = cCD_PARSER_STATE_ERROR;
						}
					} /* (memSize > 0) */
					else {
						/* Fehler bei memSize */
						ParserState = cCD_PARSER_STATE_ERROR;
					}
					break;

				/* ============================================== */
				/* DFA-Zustand: Abgleich der Datentypdefinitionen */
				/* ============================================== */
				case cCD_PARSER_STATE_COMPARE_DO_TYPE:
					iDatObjInfo.enable = TRUE;
					iDatObjInfo.pName = (unsigned long)"TypeDesc";
					DatObjInfo(&iDatObjInfo);
					if (iDatObjInfo.status == 0) {
						/* Datenmodul-Alignment beachten */
						if (iDatObjInfo.len >= (maxDbsType + 1) * sizeof(TYPE_DESC) + countDefinedItem * sizeof(ITEM_DESC) &&
							iDatObjInfo.len <  (maxDbsType + 1) * sizeof(TYPE_DESC) + countDefinedItem * sizeof(ITEM_DESC) + sizeof(unsigned long))
						{
							DbsTypeChanged = FALSE;
							pWorkTypeDesc = (TYPE_DESC*)iDatObjInfo.pDatObjMem;
							for (i=0; i<maxDbsType + 1; i++) {
								if (&pWorkTypeDesc[i] >= (TYPE_DESC*)(iDatObjInfo.pDatObjMem + iDatObjInfo.len)) {
									break;
								}
								if (pTypeDesc[i].dbsType			== pWorkTypeDesc[i].dbsType &&
									pTypeDesc[i].sizeType			== pWorkTypeDesc[i].sizeType &&
									pTypeDesc[i].sizeIntType		== pWorkTypeDesc[i].sizeIntType &&
									pTypeDesc[i].countItem			== pWorkTypeDesc[i].countItem &&
									pTypeDesc[i].countTimeItem		== pWorkTypeDesc[i].countTimeItem &&
									pTypeDesc[i].countRelatedPoints	== pWorkTypeDesc[i].countRelatedPoints
								) {
									pWorkItemDesc = pTypeDesc[i].pItemDesc;
									for (j=0; j<pTypeDesc[i].countItem; j++) {
										if (pTypeDesc[i].pItemDesc[j].offItem		== pWorkItemDesc[j].offItem &&
											pTypeDesc[i].pItemDesc[j].lenItem		== pWorkItemDesc[j].lenItem &&
											pTypeDesc[i].pItemDesc[j].sItem			== pWorkItemDesc[j].sItem &&
											pTypeDesc[i].pItemDesc[j].tsItem		== pWorkItemDesc[j].tsItem &&
											pTypeDesc[i].pItemDesc[j].idTypeItem	== pWorkItemDesc[j].idTypeItem
										) {
										}
										else {
											DbsTypeChanged = TRUE;
											break;
										}
									}
									if (DbsTypeChanged == TRUE) {
										break;
									}
								}
								else {
									DbsTypeChanged = TRUE;
									break;
								}
							}
						}
						else {
							DbsTypeChanged = TRUE;
						}
						if (DbsTypeChanged == TRUE) {
							ParserState = cCD_PARSER_STATE_DEL_DO_TYPE;
						}
						else {
							ParserState = cCD_PARSER_STATE_COUNT_DP;
						}
					}
					else if (iDatObjInfo.status == doERR_MODULNOTFOUND) {
						DbsTypeChanged = TRUE;
						ParserState = cCD_PARSER_STATE_CREATE_DO_TYPE;
					}
					else if (iDatObjInfo.status != ERR_FUB_BUSY) {
						ParserState = cCD_PARSER_STATE_ERROR;
					}
					break;

				/* ========================================================= */
				/* DFA-Zustand: Datenobjekt für Datentypdefinitionen löschen */
				/* ========================================================= */
				case cCD_PARSER_STATE_DEL_DO_TYPE:
					iDatObjDelete.enable = TRUE;
					iDatObjDelete.ident = iDatObjInfo.ident;
					DatObjDelete(&iDatObjDelete);
					if (iDatObjDelete.status == 0) {
						ParserState = cCD_PARSER_STATE_CREATE_DO_TYPE;
					}
					else if (iDatObjDelete.status != ERR_FUB_BUSY) {
						ParserState = cCD_PARSER_STATE_ERROR;
					}
					break;

				/* ========================================================= */
				/* DFA-Zustand: Datenobjekt für Datentypdefinitionen anlegen */
				/* ========================================================= */
				case cCD_PARSER_STATE_CREATE_DO_TYPE:
					iDatObjCreate.enable = TRUE;
					iDatObjCreate.grp = 0;
					iDatObjCreate.pName = (unsigned long)"TypeDesc";
					iDatObjCreate.len = (maxDbsType + 1) * sizeof(TYPE_DESC) + countDefinedItem * sizeof(ITEM_DESC);
					iDatObjCreate.MemType = doUSRRAM;
					iDatObjCreate.Option = !doNO_CS;
					iDatObjCreate.pCpyData = (unsigned long)pTypeDesc;
					DatObjCreate(&iDatObjCreate);
					if (iDatObjCreate.status == 0) {
						ParserState = cCD_PARSER_STATE_COUNT_DP;
					}
					else if (iDatObjCreate.status != ERR_FUB_BUSY) {
						ParserState = cCD_PARSER_STATE_ERROR;
					}
					break;

				/* ======================================= */
				/* DFA-Zustand: Zählen der DBS-Datenpunkte */
				/* ======================================= */
				case cCD_PARSER_STATE_COUNT_DP:
					iDatObjInfo.enable = TRUE;
					iDatObjInfo.pName = (UDINT)cKW_DBS_DM_DP_LIST;
					DatObjInfo(&iDatObjInfo);
					if (iDatObjInfo.status == 0) {
						pDA_Data = (unsigned char*)iDatObjInfo.pDatObjMem;
						SizeDA_Data = iDatObjInfo.len;

						/* go */

						/* Datenmodul von Anfang an Parsen ... */
						CountLines = 0;
						pParser = (unsigned char*)pDA_Data;

						/* Zähler rücksetzen */
						countPortData = 0;
						countTimeoutData = 0;
						countDefinedPoint = 0;
						countExistPoints = 0;
						countNotExistPoints = 0;
						countStationTypPoint = 0;
						countLogMessages = 0;
						countFubInstance = 0;

						SizeNamePoint = 0;

						/* Parser-Status loeschen */
						State_find_StationTypPoint = 0;
						State_find_Section = 0;
						State_find_Data = 0;

						/* ------ */
						/* Parsen */
						/* ------ */
						while (pParser < (unsigned char*)pDA_Data + SizeDA_Data) {

							/* Suche nach Stations/Typ/Punkt-Beschreibung */
							State_find_StationTypPoint = find_StationTypPoint(pDA_Data, pParser, pDA_Data + SizeDA_Data,
																				&pParser, &pParserLine, &pParserErr, &CountLines,
																				&pDataArg1, &SizeArg1,
																				&pDataArg2, &SizeArg2,
																				&SectionType);
							/* keine Daten oder Fehler aufgetreten ? */
							if (State_find_StationTypPoint < 0) {
								break;
							}
							else {
								countStationTypPoint++;
							}

							/* Pointer auf Station/Typ/Punkt */
							switch (SectionType) {

								/* ------------------ */
								/* Stations-Abschnitt */
								/* ------------------ */
								case cCD_STATION:
									countSection = 0;
									do {
										State_find_Section = find_Section(pDA_Data, pParser, pDA_Data + SizeDA_Data,
																			&pParser, &pParserLine, &pParserErr, &CountLines,
																			&pDataArg1, &SizeArg1,
																			&pDataArg2, &SizeArg2,
																			cKW_ALL_SECTION);
										/* keine Daten oder Fehler aufgetreten ? */
										if (State_find_Section < 0) {
											break;
										}
										else {
											countSection++;
										}

										/* Pointer auf Anfang der Sektion stellen */
										if (pDataArg2 != NULL) {
											pParser = pDataArg2;
										}
										else {
											continue;
										}

										/* alle Daten der Sektion bearbeiten */
										countData = 0;
										do {
											/* Daten der Sektion anfordern */
											State_find_Data = find_Data(pDA_Data, pParser, pDA_Data + SizeDA_Data,
																		  &pParser, &pParserLine, &pParserErr, NULL,
																		  &pDataArg1, &SizeArg1,
																		  &pDataArg2, &SizeArg2,
																		  &pDataArg3, &SizeArg3);
											/* keine Daten oder Fehler aufgetreten ? */
											if (State_find_Data < -1) {
												break;
											}
											else if (State_find_Data == -1) {
												if (pParser < (unsigned char*)pDA_Data + SizeDA_Data) {
													pParser++;
													State_find_Data = TRUE;
													continue;
												}
												else {
													break;
												}
											}
											else {
												/* Port-Bezeichner */
												if (strlen(cKW_TCP_PORT) == SizeArg1 && strncasecmp(pDataArg1, cKW_TCP_PORT, SizeArg1) == 0 &&
													strlen(cKW_TCP_PORT_NUMBER) == SizeArg2 && strncasecmp(pDataArg2, cKW_TCP_PORT_NUMBER, SizeArg2) == 0 &&
													pDataArg3 != NULL && SizeArg3 != 0 &&
													IsANumber(pDataArg3) == TRUE)
												{
													countPortData++;
												}
												/* Timeout-Bezeichner */
												else if (strlen(cKW_TCP_TIMEOUT) == SizeArg1 && strncasecmp(pDataArg1, cKW_TCP_TIMEOUT, SizeArg1) == 0 &&
													strlen(cKW_TCP_TIMEOUT_NUMBER) == SizeArg2 && strncasecmp(pDataArg2, cKW_TCP_TIMEOUT_NUMBER, SizeArg2) == 0 &&
													pDataArg3 != NULL && SizeArg3 != 0 &&
													IsANumber(pDataArg3) == TRUE)
												{
													countTimeoutData++;
												}
												/* Instanz-Anzahl */
												else if (strlen(cKW_DBS_CLIENT) == SizeArg1 && strncasecmp(pDataArg1, cKW_DBS_CLIENT, SizeArg1) == 0 &&
													strlen(cKW_DBS_CLIENT_COUNT) == SizeArg2 && strncasecmp(pDataArg2, cKW_DBS_CLIENT_COUNT, SizeArg2) == 0 &&
													pDataArg3 != NULL && SizeArg3 != 0 &&
													IsANumber(pDataArg3) == TRUE)
												{
													countEventInstance = atoi(pDataArg3);
												}
												/* Applikation-Anzahl */
												else if (strlen(cKW_DBS_APP) == SizeArg1 && strncasecmp(pDataArg1, cKW_DBS_APP, SizeArg1) == 0 &&
													strlen(cKW_DBS_APP_COUNT) == SizeArg2 && strncasecmp(pDataArg2, cKW_DBS_APP_COUNT, SizeArg2) == 0 &&
													pDataArg3 != NULL && SizeArg3 != 0 &&
													IsANumber(pDataArg3) == TRUE)
												{
													countWriteInstance = atoi(pDataArg3);
												}
												/* Anlagen-Bezeichner */
												else if (strlen(cKW_DBS_UNIT) == SizeArg1 && strncasecmp(pDataArg1, cKW_DBS_UNIT, SizeArg1) == 0 &&
													strlen(cKW_DBS_UNIT_NUMBER) == SizeArg2 && strncasecmp(pDataArg2, cKW_DBS_UNIT_NUMBER, SizeArg2) == 0 &&
													pDataArg3 != NULL && SizeArg3 != 0 &&
													IsANumber(pDataArg3) == TRUE)
												{
													countUnitData++;
													DbsUnit = atoi(pDataArg3);
													maxDbsUnit = (DbsUnit > maxDbsUnit) ? DbsUnit : maxDbsUnit;
												}
												/* Datenpunkt-Bezeichner */
												else if (strlen(cKW_DBS_POINT) == SizeArg1 && strncasecmp(pDataArg1, cKW_DBS_POINT, SizeArg1) == 0 &&
													strlen(cKW_DBS_POINT_NUMBER) == SizeArg2 && strncasecmp(pDataArg2, cKW_DBS_POINT_NUMBER, SizeArg2) == 0 &&
													pDataArg3 != NULL && SizeArg3 != 0 &&
													IsANumber(pDataArg3) == TRUE)
												{
													countPointData++;
												}
												/* unbekannte Zuweisung */
												else {
												}
											}
										} while (State_find_Data == TRUE);
									} while (State_find_Section == TRUE);
									break;

								/* ------------------- */
								/* Typ/Block-Abschnitt */
								/* ------------------- */
								case cCD_TYP:
									countSection = 0;
									do {
										State_find_Section = find_Section(pDA_Data, pParser, pDA_Data + SizeDA_Data,
																			&pParser, &pParserLine, &pParserErr, &CountLines,
																			&pDataArg1, &SizeArg1,
																			&pDataArg2, &SizeArg2,
																			cKW_TCP_SECTION);
										/* keine Daten oder Fehler aufgetreten ? */
										if (State_find_Section < 0) {
											break;
										}
										else {
											countSection++;
										}

										/* Pointer auf Anfang der Sektion stellen */
										if (pDataArg2 != NULL) {
											pParser = pDataArg2;
										}
										else {
											continue;
										}

										/* alle Daten der Sektion bearbeiten */
										countData = 0;
										do {
											/* Daten der Sektion anfordern */
											State_find_Data = find_Data(pDA_Data, pParser, pDA_Data + SizeDA_Data,
																		  &pParser, &pParserLine, &pParserErr, NULL,
																		  &pDataArg1, &SizeArg1,
																		  &pDataArg2, &SizeArg2,
																		  &pDataArg3, &SizeArg3);
											/* keine Daten oder Fehler aufgetreten ? */
											if (State_find_Data < 0) {
												break;
											}
											else {
												/* Port-Bezeichner */
												if (strlen(cKW_TCP_PORT) == SizeArg1 && strncasecmp(pDataArg1, cKW_TCP_PORT, SizeArg1) == 0 &&
													strlen(cKW_TCP_PORT_NUMBER) == SizeArg2 && strncasecmp(pDataArg2, cKW_TCP_PORT_NUMBER, SizeArg2) == 0 &&
													pDataArg3 != NULL && SizeArg3 != 0 &&
													IsANumber(pDataArg3) == TRUE)
												{
													countPortData++;
												}
												/* Timeout-Bezeichner */
												else if (strlen(cKW_TCP_TIMEOUT) == SizeArg1 && strncasecmp(pDataArg1, cKW_TCP_TIMEOUT, SizeArg1) == 0 &&
													strlen(cKW_TCP_TIMEOUT_NUMBER) == SizeArg2 && strncasecmp(pDataArg2, cKW_TCP_TIMEOUT_NUMBER, SizeArg2) == 0 &&
													pDataArg3 != NULL && SizeArg3 != 0 &&
													IsANumber(pDataArg3) == TRUE)
												{
													countTimeoutData++;
												}
												/* Anlagen-Bezeichner */
												else if (strlen(cKW_DBS_UNIT) == SizeArg1 && strncasecmp(pDataArg1, cKW_DBS_UNIT, SizeArg1) == 0 &&
													strlen(cKW_DBS_UNIT_NUMBER) == SizeArg2 && strncasecmp(pDataArg2, cKW_DBS_UNIT_NUMBER, SizeArg2) == 0 &&
													pDataArg3 != NULL && SizeArg3 != 0 &&
													IsANumber(pDataArg3) == TRUE)
												{
													countUnitData++;
													DbsUnit = atoi(pDataArg3);
													maxDbsUnit = (DbsUnit > maxDbsUnit) ? DbsUnit : maxDbsUnit;
												}
												/* Datenpunkt-Bezeichner */
												else if (strlen(cKW_DBS_POINT) == SizeArg1 && strncasecmp(pDataArg1, cKW_DBS_POINT, SizeArg1) == 0 &&
													strlen(cKW_DBS_POINT_NUMBER) == SizeArg2 && strncasecmp(pDataArg2, cKW_DBS_POINT_NUMBER, SizeArg2) == 0 &&
													pDataArg3 != NULL && SizeArg3 != 0 &&
													IsANumber(pDataArg3) == TRUE)
												{
													countPointData++;
												}
												/* unbekannte Zuweisung */
												else {
												}
											}
										} while (State_find_Data == TRUE);
									} while (State_find_Section == TRUE);
									break;

								/* -------------------- */
								/* Datenpunkt-Abschnitt */
								/* -------------------- */
								case cCD_POINT:

									/* Datenpunkt feststellen */
									StateGetDpInfo = GetDpInfo(pDataArg1, &DtIdx, &DpIdx, NULL);
									StateGetDpInfo = 1;
									flagDbsPoint = FALSE;
									flagDbsType = FALSE;
									flagDbsUnit = FALSE;
									flagDbsFub = FALSE;
									countPointData = 0;
									countSection = 0;
									SizeNamePoint += SizeArg1 + 1;
									do {
										State_find_Section = find_Section(pDA_Data, pParser, pDA_Data + SizeDA_Data,
																			&pParser, &pParserLine, &pParserErr, &CountLines,
																			&pDataArg1, &SizeArg1,
																			&pDataArg2, &SizeArg2,
																			cKW_ALL_SECTION);
										/* keine Daten oder Fehler aufgetreten ? */
										if (State_find_Section < 0) {
											break;
										}
										else {
											countSection++;
										}

										/* Pointer auf Anfang der Sektion stellen */
										if (pDataArg2 != NULL) {
											pParser = pDataArg2;
										}
										else {
											continue;
										}

										/* alle Daten der Sektion bearbeiten */
										do {
											/* Daten der Sektion anfordern */
											State_find_Data = find_Data(pDA_Data, pParser, pDA_Data + SizeDA_Data,
																		  &pParser, &pParserLine, &pParserErr, NULL,
																		  &pDataArg1, &SizeArg1,
																		  &pDataArg2, &SizeArg2,
																		  &pDataArg3, &SizeArg3);
											/* keine Daten oder Fehler aufgetreten ? */
											if (State_find_Data < 0) {
												break;
											}
											else {
												/* Port-Bezeichner */
												if (strlen(cKW_TCP_PORT) == SizeArg1 && strncasecmp(pDataArg1, cKW_TCP_PORT, SizeArg1) == 0 &&
													strlen(cKW_TCP_PORT_NUMBER) == SizeArg2 && strncasecmp(pDataArg2, cKW_TCP_PORT_NUMBER, SizeArg2) == 0 &&
													pDataArg3 != NULL && SizeArg3 != 0 &&
													IsANumber(pDataArg3) == TRUE)
												{
													countPortData++;
												}
												/* Timeout-Bezeichner */
												else if (strlen(cKW_TCP_TIMEOUT) == SizeArg1 && strncasecmp(pDataArg1, cKW_TCP_TIMEOUT, SizeArg1) == 0 &&
													strlen(cKW_TCP_TIMEOUT_NUMBER) == SizeArg2 && strncasecmp(pDataArg2, cKW_TCP_TIMEOUT_NUMBER, SizeArg2) == 0 &&
													pDataArg3 != NULL && SizeArg3 != 0 &&
													IsANumber(pDataArg3) == TRUE)
												{
													countTimeoutData++;
												}
												/* Anlagen-Bezeichner */
												else if (strlen(cKW_DBS_UNIT) == SizeArg1 && strncasecmp(pDataArg1, cKW_DBS_UNIT, SizeArg1) == 0 &&
													strlen(cKW_DBS_UNIT_NUMBER) == SizeArg2 && strncasecmp(pDataArg2, cKW_DBS_UNIT_NUMBER, SizeArg2) == 0 &&
													pDataArg3 != NULL && SizeArg3 != 0 &&
													IsANumber(pDataArg3) == TRUE)
												{
													countUnitData++;
													DbsUnit = atoi(pDataArg3);
													maxDbsUnit = (DbsUnit > maxDbsUnit) ? DbsUnit : maxDbsUnit;
													flagDbsUnit = TRUE;
												}
												/* Datentyp-Bezeichner */
												else if (strlen(cKW_DBS_TYPE) == SizeArg1 && strncasecmp(pDataArg1, cKW_DBS_TYPE, SizeArg1) == 0 &&
													pDataArg3 != NULL && SizeArg3 != 0)
												{
													flagDbsType = FALSE;
													for (i=0; i<=maxDbsType; i++) {
														if (pTypeDesc[i].pTypeName != NULL) {
															if (strncmp(pDataArg3, pTypeDesc[i].pTypeName, SizeArg3) == 0 &&
																strlen(pTypeDesc[i].pTypeName) == SizeArg3)
															{
																DbsType = i;
																flagDbsType = TRUE;
																break;
															}
														}
													}
													if (flagDbsType == FALSE) {
													}
													else {
													}
												}
												/* Datenpunkt-Bezeichner */
												else if (strlen(cKW_DBS_POINT) == SizeArg1 && strncasecmp(pDataArg1, cKW_DBS_POINT, SizeArg1) == 0 &&
													strlen(cKW_DBS_POINT_NUMBER) == SizeArg2 && strncasecmp(pDataArg2, cKW_DBS_POINT_NUMBER, SizeArg2) == 0 &&
													pDataArg3 != NULL && SizeArg3 != 0 &&
													IsANumber(pDataArg3) == TRUE)
												{
													DbsPoint = atoi(pDataArg3);
													flagDbsPoint = TRUE;
													if (countPointData == 0) {
														countPointData++;
														if (StateGetDpInfo == 1) {
															countDefinedPoint++;
															countExistPoints++;
														}
														else {
															countNotExistPoints++;
														}
													}
													else {
														/* Warnung: wiederholte Dp-Definition */
													}
												}
												/* Fub-Instanz-Bezeichner */
												else if (strlen(cKW_DBS_FUB) == SizeArg1 && strncasecmp(pDataArg1, cKW_DBS_FUB, SizeArg1) == 0 &&
													pDataArg3 != NULL && SizeArg3 != 0 &&
													IsANumber(pDataArg3) == TRUE)
												{
													countFub++;
													if (atoi(pDataArg3) == 1) {
														flagDbsFub = TRUE;
													}
												}
												/* unbekannte Zuweisung */
												else {
												}
											}
										} while (State_find_Data == TRUE);
									} while (State_find_Section == TRUE);
									if (flagDbsUnit == TRUE && flagDbsType == TRUE && flagDbsPoint == TRUE && flagDbsFub == TRUE) {
										countFubInstance += pTypeDesc[DbsType].countItem;
									}
									break;
							} /* (SectionType) */
						} /* (pParser < (unsigned char*)pDA_Data + SizeDA_Data) */

						/* ---------------- */
						/* nächster Zustand */
						/* ---------------- */
						ParserState = cCD_PARSER_STATE_DEF_DP;

					} /* (DA_DataOk == TRUE) */
					else {
						/* Fehler beim Datenmodul */
						ErrStatistics("dbserv", ERRLOG, EC_DA_NOT_FOUND + EC_DBS_BASE, CountLines, ERR_DBS_PRE, ET_DA_NOT_FOUND);
						ParserState = cCD_PARSER_STATE_ERROR;
					}
					break;

				/* ===================================================================== */
				/* DFA-Zustand: Speicher allokieren und Aufbau der Bäume für Datenpunkte */
				/* ===================================================================== */
				case cCD_PARSER_STATE_DEF_DP:

					maxUsedUnit = maxDbsUnit;
					maxUsedType = maxDbsType;

					/* ----------------------------------------- */
					/* Baum Unit -> Type aufbauen (Wurzelknoten) */
					/* ----------------------------------------- */
					memSize = (maxUsedUnit + 1) * sizeof(ACCESS_UNIT);
					StateTMP_alloc = TMP_alloc(memSize, (void*)&pAccessUnit);
					if (StateTMP_alloc == 0) {
						SmemSize += 0;
						StmpSize += memSize;
						memset(pAccessUnit, 0, memSize);

						memSize = countDefinedPoint * sizeof(POINT_DESC) + SizeNamePoint;
						StateTMP_alloc = TMP_alloc(memSize, (void*)&pPointDesc);
						if (StateTMP_alloc == 0) {
							SmemSize += 0;
							StmpSize += memSize;
							memset(pPointDesc, 0, memSize);
							pWorkPointName = (unsigned char*)(pPointDesc + countDefinedPoint);

							memSize = countFubInstance * sizeof(FUB_DESC);
							StateTMP_alloc = TMP_alloc(memSize, (void*)&pFubInstanceDesc);
							if (StateTMP_alloc == 0) {
								SmemSize += 0;
								StmpSize += memSize;
								memset(pFubInstanceDesc, 0, memSize);

								/* Datenmodul von Anfang an Parsen ... */
								CountLines = 0;
								pParser = (unsigned char*)pDA_Data;

								/* Zähler rücksetzen */
								countPortData = 0;
								countTimeoutData = 0;
								countDefinedPoint = 0;
								countExistPoints = 0;
								countNotExistPoints = 0;

								countNotDefinedItems = 0;
								countInvalidExistItems = 0;
								countNotExistItems = 0;

								countStationTypPoint = 0;
								countLogMessages = 0;
								countFubInstance = 0;

								/* Parser-Status loeschen */
								State_find_StationTypPoint = 0;
								State_find_Section = 0;
								State_find_Data = 0;

								/* ------ */
								/* Parsen */
								/* ------ */
								while (pParser < (unsigned char*)pDA_Data + SizeDA_Data) {

									/* Suche nach Stations/Typ/Punkt-Beschreibung */
									State_find_StationTypPoint = find_StationTypPoint(pDA_Data, pParser, pDA_Data + SizeDA_Data,
																						&pParser, &pParserLine, &pParserErr, &CountLines,
																						&pDataArg1, &SizeArg1,
																						&pDataArg2, &SizeArg2,
																						&SectionType);
									/* keine Daten oder Fehler aufgetreten ? */
									if (State_find_StationTypPoint < 0) {
										break;
									}
									else {
										countStationTypPoint++;
									}

									/* Pointer auf Station/Typ/Punkt */
									switch (SectionType) {

										/* ------------------ */
										/* Stations-Abschnitt */
										/* ------------------ */
										case cCD_STATION:
											countSection = 0;
											do {
												State_find_Section = find_Section(pDA_Data, pParser, pDA_Data + SizeDA_Data,
																					&pParser, &pParserLine, &pParserErr, &CountLines,
																					&pDataArg1, &SizeArg1,
																					&pDataArg2, &SizeArg2,
																					cKW_TCP_SECTION);
												/* keine Daten oder Fehler aufgetreten ? */
												if (State_find_Section < 0) {
													break;
												}
												else {
													countSection++;
												}

												/* Pointer auf Anfang der Sektion stellen */
												if (pDataArg2 != NULL) {
													pParser = pDataArg2;
												}
												else {
													continue;
												}

												/* alle Daten der Sektion bearbeiten */
												countData = 0;
												do {
													/* Daten der Sektion anfordern */
													State_find_Data = find_Data(pDA_Data, pParser, pDA_Data + SizeDA_Data,
																				  &pParser, &pParserLine, &pParserErr, NULL,
																				  &pDataArg1, &SizeArg1,
																				  &pDataArg2, &SizeArg2,
																				  &pDataArg3, &SizeArg3);
													/* keine Daten oder Fehler aufgetreten ? */
													if (State_find_Data < 0) {
														break;
													}
													else {
														/* Port-Bezeichner */
														if (strlen(cKW_TCP_PORT) == SizeArg1 && strncasecmp(pDataArg1, cKW_TCP_PORT, SizeArg1) == 0 &&
															strlen(cKW_TCP_PORT_NUMBER) == SizeArg2 && strncasecmp(pDataArg2, cKW_TCP_PORT_NUMBER, SizeArg2) == 0 &&
															pDataArg3 != NULL && SizeArg3 != 0 &&
															IsANumber(pDataArg3) == TRUE)
														{
															countPortData++;
														}
														/* Timeout-Bezeichner */
														else if (strlen(cKW_TCP_TIMEOUT) == SizeArg1 && strncasecmp(pDataArg1, cKW_TCP_TIMEOUT, SizeArg1) == 0 &&
															strlen(cKW_TCP_TIMEOUT_NUMBER) == SizeArg2 && strncasecmp(pDataArg2, cKW_TCP_TIMEOUT_NUMBER, SizeArg2) == 0 &&
															pDataArg3 != NULL && SizeArg3 != 0 &&
															IsANumber(pDataArg3) == TRUE)
														{
															countTimeoutData++;
														}
														/* Anlagen-Bezeichner */
														else if (strlen(cKW_DBS_UNIT) == SizeArg1 && strncasecmp(pDataArg1, cKW_DBS_UNIT, SizeArg1) == 0 &&
															strlen(cKW_DBS_UNIT_NUMBER) == SizeArg2 && strncasecmp(pDataArg2, cKW_DBS_UNIT_NUMBER, SizeArg2) == 0 &&
															pDataArg3 != NULL && SizeArg3 != 0 &&
															IsANumber(pDataArg3) == TRUE)
														{
															countUnitData++;
															DbsUnit = atoi(pDataArg3);
															maxDbsUnit = (DbsUnit > maxDbsUnit) ? DbsUnit : maxDbsUnit;
														}
														/* Datenpunkt-Bezeichner */
														else if (strlen(cKW_DBS_POINT) == SizeArg1 && strncasecmp(pDataArg1, cKW_DBS_POINT, SizeArg1) == 0 &&
															strlen(cKW_DBS_POINT_NUMBER) == SizeArg2 && strncasecmp(pDataArg2, cKW_DBS_POINT_NUMBER, SizeArg2) == 0 &&
															pDataArg3 != NULL && SizeArg3 != 0 &&
															IsANumber(pDataArg3) == TRUE)
														{
															countPointData++;
														}
														/* unbekannte Zuweisung */
														else {
														}
													}
												} while (State_find_Data == TRUE);
											} while (State_find_Section == TRUE);
											break;

										/* ------------------- */
										/* Typ/Block-Abschnitt */
										/* ------------------- */
										case cCD_TYP:
											countSection = 0;
											do {
												State_find_Section = find_Section(pDA_Data, pParser, pDA_Data + SizeDA_Data,
																					&pParser, &pParserLine, &pParserErr, &CountLines,
																					&pDataArg1, &SizeArg1,
																					&pDataArg2, &SizeArg2,
																					cKW_TCP_SECTION);
												/* keine Daten oder Fehler aufgetreten ? */
												if (State_find_Section < 0) {
													break;
												}
												else {
													countSection++;
												}

												/* Pointer auf Anfang der Sektion stellen */
												if (pDataArg2 != NULL) {
													pParser = pDataArg2;
												}
												else {
													continue;
												}

												/* alle Daten der Sektion bearbeiten */
												countData = 0;
												do {
													/* Daten der Sektion anfordern */
													State_find_Data = find_Data(pDA_Data, pParser, pDA_Data + SizeDA_Data,
																				  &pParser, &pParserLine, &pParserErr, NULL,
																				  &pDataArg1, &SizeArg1,
																				  &pDataArg2, &SizeArg2,
																				  &pDataArg3, &SizeArg3);
													/* keine Daten oder Fehler aufgetreten ? */
													if (State_find_Data < 0) {
														break;
													}
													else {
														/* Port-Bezeichner */
														if (strlen(cKW_TCP_PORT) == SizeArg1 && strncasecmp(pDataArg1, cKW_TCP_PORT, SizeArg1) == 0 &&
															strlen(cKW_TCP_PORT_NUMBER) == SizeArg2 && strncasecmp(pDataArg2, cKW_TCP_PORT_NUMBER, SizeArg2) == 0 &&
															pDataArg3 != NULL && SizeArg3 != 0 &&
															IsANumber(pDataArg3) == TRUE)
														{
															countPortData++;
														}
														/* Timeout-Bezeichner */
														else if (strlen(cKW_TCP_TIMEOUT) == SizeArg1 && strncasecmp(pDataArg1, cKW_TCP_TIMEOUT, SizeArg1) == 0 &&
															strlen(cKW_TCP_TIMEOUT_NUMBER) == SizeArg2 && strncasecmp(pDataArg2, cKW_TCP_TIMEOUT_NUMBER, SizeArg2) == 0 &&
															pDataArg3 != NULL && SizeArg3 != 0 &&
															IsANumber(pDataArg3) == TRUE)
														{
															countTimeoutData++;
														}
														/* Anlagen-Bezeichner */
														else if (strlen(cKW_DBS_UNIT) == SizeArg1 && strncasecmp(pDataArg1, cKW_DBS_UNIT, SizeArg1) == 0 &&
															strlen(cKW_DBS_UNIT_NUMBER) == SizeArg2 && strncasecmp(pDataArg2, cKW_DBS_UNIT_NUMBER, SizeArg2) == 0 &&
															pDataArg3 != NULL && SizeArg3 != 0 &&
															IsANumber(pDataArg3) == TRUE)
														{
															countUnitData++;
															DbsUnit = atoi(pDataArg3);
															maxDbsUnit = (DbsUnit > maxDbsUnit) ? DbsUnit : maxDbsUnit;
														}
														/* Datenpunkt-Bezeichner */
														else if (strlen(cKW_DBS_POINT) == SizeArg1 && strncasecmp(pDataArg1, cKW_DBS_POINT, SizeArg1) == 0 &&
															strlen(cKW_DBS_POINT_NUMBER) == SizeArg2 && strncasecmp(pDataArg2, cKW_DBS_POINT_NUMBER, SizeArg2) == 0 &&
															pDataArg3 != NULL && SizeArg3 != 0 &&
															IsANumber(pDataArg3) == TRUE)
														{
															countPointData++;
														}
														/* unbekannte Zuweisung */
														else {
														}
													}
												} while (State_find_Data == TRUE);
											} while (State_find_Section == TRUE);
											break;

										/* -------------------- */
										/* Datenpunkt-Abschnitt */
										/* -------------------- */
										case cCD_POINT:

											/* Datenpunkt feststellen */
											pPointName = pDataArg1, lenPointName = SizeArg1;
											flagDbsPoint = FALSE;
											flagDbsType = FALSE;
											flagDbsUnit = FALSE;
											flagDbsFub = FALSE;
											countPointData = 0;
											countSection = 0;
											do {
												State_find_Section = find_Section(pDA_Data, pParser, pDA_Data + SizeDA_Data,
																					&pParser, &pParserLine, &pParserErr, &CountLines,
																					&pDataArg1, &SizeArg1,
																					&pDataArg2, &SizeArg2,
																					cKW_ALL_SECTION);
												/* keine Daten oder Fehler aufgetreten ? */
												if (State_find_Section < 0) {
													break;
												}
												else {
													countSection++;
												}

												/* Pointer auf Anfang der Sektion stellen */
												if (pDataArg2 != NULL) {
													pParser = pDataArg2;
												}
												else {
													continue;
												}

												/* alle Daten der Sektion bearbeiten */
												do {
													/* Daten der Sektion anfordern */
													State_find_Data = find_Data(pDA_Data, pParser, pDA_Data + SizeDA_Data,
																				  &pParser, &pParserLine, &pParserErr, NULL,
																				  &pDataArg1, &SizeArg1,
																				  &pDataArg2, &SizeArg2,
																				  &pDataArg3, &SizeArg3);
													/* keine Daten oder Fehler aufgetreten ? */
													if (State_find_Data < 0) {
														break;
													}
													else {
														/* Port-Bezeichner */
														if (strlen(cKW_TCP_PORT) == SizeArg1 && strncasecmp(pDataArg1, cKW_TCP_PORT, SizeArg1) == 0 &&
															strlen(cKW_TCP_PORT_NUMBER) == SizeArg2 && strncasecmp(pDataArg2, cKW_TCP_PORT_NUMBER, SizeArg2) == 0 &&
															pDataArg3 != NULL && SizeArg3 != 0 &&
															IsANumber(pDataArg3) == TRUE)
														{
															countPortData++;
														}
														/* Timeout-Bezeichner */
														else if (strlen(cKW_TCP_TIMEOUT) == SizeArg1 && strncasecmp(pDataArg1, cKW_TCP_TIMEOUT, SizeArg1) == 0 &&
															strlen(cKW_TCP_TIMEOUT_NUMBER) == SizeArg2 && strncasecmp(pDataArg2, cKW_TCP_TIMEOUT_NUMBER, SizeArg2) == 0 &&
															pDataArg3 != NULL && SizeArg3 != 0 &&
															IsANumber(pDataArg3) == TRUE)
														{
															countTimeoutData++;
														}
														/* Anlagen-Bezeichner */
														else if (strlen(cKW_DBS_UNIT) == SizeArg1 && strncasecmp(pDataArg1, cKW_DBS_UNIT, SizeArg1) == 0 &&
															strlen(cKW_DBS_UNIT_NUMBER) == SizeArg2 && strncasecmp(pDataArg2, cKW_DBS_UNIT_NUMBER, SizeArg2) == 0 &&
															pDataArg3 != NULL && SizeArg3 != 0 &&
															IsANumber(pDataArg3) == TRUE)
														{
															countUnitData++;
															if (atoi(pDataArg3) >= 0 && atoi(pDataArg3) <= cMAX_UNIT_DEF) {
																DbsUnit = atoi(pDataArg3);
																maxDbsUnit = (DbsUnit > maxDbsUnit) ? DbsUnit : maxDbsUnit;
																flagDbsUnit = TRUE;
															}
															else {
															}
														}
														/* Datentyp-Bezeichner */
														else if (strlen(cKW_DBS_TYPE) == SizeArg1 && strncasecmp(pDataArg1, cKW_DBS_TYPE, SizeArg1) == 0 &&
															pDataArg3 != NULL && SizeArg3 != 0)
														{
															flagDbsType = FALSE;
															for (i=0; i<=maxDbsType; i++) {
																if (pTypeDesc[i].pTypeName != NULL) {
																	if (strncmp(pDataArg3, pTypeDesc[i].pTypeName, SizeArg3) == 0 &&
																		strlen(pTypeDesc[i].pTypeName) == SizeArg3)
																	{
																		DbsType = i;
																		flagDbsType = TRUE;
																		break;
																	}
																}
															}
															if (flagDbsType == FALSE) {
															}
															else {
															}
														}
														/* Datenpunkt-Bezeichner */
														else if (strlen(cKW_DBS_POINT) == SizeArg1 && strncasecmp(pDataArg1, cKW_DBS_POINT, SizeArg1) == 0 &&
															strlen(cKW_DBS_POINT_NUMBER) == SizeArg2 && strncasecmp(pDataArg2, cKW_DBS_POINT_NUMBER, SizeArg2) == 0 &&
															pDataArg3 != NULL && SizeArg3 != 0 &&
															IsANumber(pDataArg3) == TRUE)
														{
															if (countPointData == 0) {
																countPointData++;
																if (atoi(pDataArg3) >= 0 && atoi(pDataArg3) <= cMAX_POINT_DEF) {
																	DbsPoint = atoi(pDataArg3);
																	pTempData = pDataArg3;
																	flagDbsPoint = TRUE;
																	/*if (StateGetDpInfo == 1) {
																		countExistPoints++;
																	}
																	else {
																		countNotExistPoints++;
																	}*/
																}
																else {
																}
															}
															else {
																/* Warnung: wiederholte Dp-Definition */
															}
														}
														/* Fub-Instanz-Bezeichner */
														else if (strlen(cKW_DBS_FUB) == SizeArg1 && strncasecmp(pDataArg1, cKW_DBS_FUB, SizeArg1) == 0 &&
															pDataArg3 != NULL && SizeArg3 != 0 &&
															IsANumber(pDataArg3) == TRUE)
														{
															countFub++;
															if (atoi(pDataArg3) == 1) {
																flagDbsFub = TRUE;
															}
														}
														/* unbekannte Zuweisung */
														else {
														}
													}
												} while (State_find_Data == TRUE);
											} while (State_find_Section == TRUE);
											if (flagDbsUnit == TRUE && flagDbsType == TRUE && flagDbsPoint == TRUE) {
												maxUsedUnit = (maxUsedUnit > DbsUnit) ? maxUsedUnit : DbsUnit;
												maxUsedType = (maxUsedType > DbsType) ? maxUsedType : DbsType;

												/* Datenpunkt eindeutig ? */
												flag = FALSE;
												for (i=0; i<countDefinedPoint; i++) {
													if (pPointDesc[i].pPointName != NULL) {
														if (strlen(pPointDesc[i].pPointName) == lenPointName &&
															strncmp(pPointDesc[i].pPointName, pPointName, strlen(pPointDesc[i].pPointName)) == 0)
														{
															flag = TRUE;
															break;
														}
													}
													if (pPointDesc[i].dbsUnit == DbsUnit &&
														pPointDesc[i].dbsType == DbsType &&
														pPointDesc[i].dbsPoint == DbsPoint)
													{
														flag = TRUE;
														break;
													}
												} /* (i=0; i<countDefinedPoint; i++) */
												if (flag == FALSE) {
													if (pPointDesc[countDefinedPoint].pPointName == NULL) {
														pPointDesc[countDefinedPoint].pPointName = pWorkPointName;
													}
													strncpy(pPointDesc[countDefinedPoint].pPointName, pPointName, lenPointName);
													pWorkPointName = pWorkPointName + lenPointName + 1;
												}
												else {
													/* wiederholte Datenpunkt definition */
													/* !!! CHECK !!! */
													strcat(strcat(strcpy(logBuffer, (char*)iDatObjInfo.pName), ET_POINT_ALREADY_EXIST), "\n");
													strcat(strncat(logBuffer, pPointName, lenPointName), "\n");
													strncat(logBuffer, pDataArg1, pDataArg3 - pDataArg1 + SizeArg3);
													ErrStatistics("dbserv", ERRLOG, EC_POINT_ALREADY_EXIST + EC_DBS_BASE, CountLines, ERR_DBS_PRE, logBuffer);
												}

												/* Datenpunkt-Deskriptor aufbauen */
												pPointDesc[countDefinedPoint].dbsUnit  = DbsUnit;
												pPointDesc[countDefinedPoint].dbsType  = DbsType;
												pPointDesc[countDefinedPoint].dbsPoint = DbsPoint;
												countDefinedPoint++;

												/* Wurzelknoten für Datentypen aufbauen */
												pAccessUnit[DbsUnit].countType = (DbsType + 1 > pAccessUnit[DbsUnit].countType) ? DbsType + 1 : pAccessUnit[DbsUnit].countType;

												/* Fub-Instanz */
												if (flagDbsFub == TRUE) {
													flagDbsExistPoints = FALSE;
													flagDbsNotExistPoints = FALSE;
													for (i=0; i<pTypeDesc[DbsType].countItem; i++) {
														strncpy(PointName, pPointName, sizeof(PointName));
														/* Namen über Item-Namen zusammensetzen */
														flagDbsFubInstance = TRUE;
														if (pTypeDesc[DbsType].countItem > 1) {
															if (pTypeDesc[DbsType].pItemDesc[i].pNameItem != NULL) {
																if (sizeof(PointName) - strlen(PointName) > strlen(pTypeDesc[DbsType].pItemDesc[i].pNameItem)) {
																	strcat(PointName, pTypeDesc[DbsType].pItemDesc[i].pNameItem);
																}
															}
															else {
																/* kein Itemname angegeben */
																countNotDefinedItems++;
																flagDbsFubInstance = FALSE;
															}
														}
														stateFubInstance = PV_xgetadr(PointName, &pFubInstance, &lenFubInstance);
														if (flagDbsFubInstance == FALSE) {
															if (stateFubInstance == 0) {
																countInvalidExistItems++;
																if (flagDbsExistPoints == FALSE) {
																	flagDbsExistPoints = TRUE;
																	countExistPoints++;
																}
															}
															else {
																/*countNotExistItems++;
																if (flagDbsNotExistPoints == FALSE) {
																	flagDbsNotExistPoints = TRUE;
																	countNotExistPoints++;
																}*/
															}
														}
														else {
															if (stateFubInstance == 0) {
																if (pTypeDesc[DbsType].pItemDesc[i].idTypeItem == cDBS_IDTYPE_BOOL &&
																	pTypeDesc[DbsType].pItemDesc[i].tsItem == FALSE)
																{
																	((DbsBool_typ*)pFubInstance)->SetValue = TRUE;

																	((DbsBool_typ*)pFubInstance)->FubRef.dbsUnit = DbsUnit;
																	((DbsBool_typ*)pFubInstance)->FubRef.dbsDevice = cDBS_DEFAULT_DEVICE;
																	((DbsBool_typ*)pFubInstance)->FubRef.dbsType = DbsType;
																	((DbsBool_typ*)pFubInstance)->FubRef.dbsPoint = DbsPoint;
																	((DbsBool_typ*)pFubInstance)->FubRef.dbsItem = i;
																	((DbsBool_typ*)pFubInstance)->FubRef.countItem = pTypeDesc[DbsType].countItem;
																	((DbsBool_typ*)pFubInstance)->FubRef.pidBrServer = 1;
																	((DbsBool_typ*)pFubInstance)->FubRef.this = pFubInstance;

																	pFubInstanceDesc[countFubInstance].dbsUnit = DbsUnit;
																	pFubInstanceDesc[countFubInstance].dbsType = DbsType;
																	pFubInstanceDesc[countFubInstance].dbsPoint = DbsPoint;
																	pFubInstanceDesc[countFubInstance].dbsItem = i;
																	pFubInstanceDesc[countFubInstance].pFubInstance = (unsigned char*)pFubInstance;
																	countFubInstance++;
																}
																else if (pTypeDesc[DbsType].pItemDesc[i].idTypeItem == cDBS_IDTYPE_BOOL &&
																	pTypeDesc[DbsType].pItemDesc[i].tsItem == TRUE)
																{
																	((DbsBoolTs_typ*)pFubInstance)->SetValue = TRUE;

																	((DbsBoolTs_typ*)pFubInstance)->FubRef.dbsUnit = DbsUnit;
																	((DbsBoolTs_typ*)pFubInstance)->FubRef.dbsDevice = cDBS_DEFAULT_DEVICE;
																	((DbsBoolTs_typ*)pFubInstance)->FubRef.dbsType = DbsType;
																	((DbsBoolTs_typ*)pFubInstance)->FubRef.dbsPoint = DbsPoint;
																	((DbsBoolTs_typ*)pFubInstance)->FubRef.dbsItem = i;
																	((DbsBoolTs_typ*)pFubInstance)->FubRef.countItem = pTypeDesc[DbsType].countItem;
																	((DbsBoolTs_typ*)pFubInstance)->FubRef.pidBrServer = 1;
																	((DbsBoolTs_typ*)pFubInstance)->FubRef.this = pFubInstance;

																	pFubInstanceDesc[countFubInstance].dbsUnit = DbsUnit;
																	pFubInstanceDesc[countFubInstance].dbsType = DbsType;
																	pFubInstanceDesc[countFubInstance].dbsPoint = DbsPoint;
																	pFubInstanceDesc[countFubInstance].dbsItem = i;
																	pFubInstanceDesc[countFubInstance].pFubInstance = (unsigned char*)pFubInstance;
																	countFubInstance++;
																}
																else if (pTypeDesc[DbsType].pItemDesc[i].idTypeItem == cDBS_IDTYPE_USINT &&
																	pTypeDesc[DbsType].pItemDesc[i].tsItem == FALSE)
																{
																	((DbsUsint_typ*)pFubInstance)->SetValue = TRUE;

																	((DbsUsint_typ*)pFubInstance)->FubRef.dbsUnit = DbsUnit;
																	((DbsUsint_typ*)pFubInstance)->FubRef.dbsDevice = cDBS_DEFAULT_DEVICE;
																	((DbsUsint_typ*)pFubInstance)->FubRef.dbsType = DbsType;
																	((DbsUsint_typ*)pFubInstance)->FubRef.dbsPoint = DbsPoint;
																	((DbsUsint_typ*)pFubInstance)->FubRef.dbsItem = i;
																	((DbsUsint_typ*)pFubInstance)->FubRef.countItem = pTypeDesc[DbsType].countItem;
																	((DbsUsint_typ*)pFubInstance)->FubRef.pidBrServer = 1;
																	((DbsUsint_typ*)pFubInstance)->FubRef.this = pFubInstance;

																	pFubInstanceDesc[countFubInstance].dbsUnit = DbsUnit;
																	pFubInstanceDesc[countFubInstance].dbsType = DbsType;
																	pFubInstanceDesc[countFubInstance].dbsPoint = DbsPoint;
																	pFubInstanceDesc[countFubInstance].dbsItem = i;
																	pFubInstanceDesc[countFubInstance].pFubInstance = (unsigned char*)pFubInstance;
																	countFubInstance++;
																}
																else if (pTypeDesc[DbsType].pItemDesc[i].idTypeItem == cDBS_IDTYPE_USINT &&
																	pTypeDesc[DbsType].pItemDesc[i].tsItem == TRUE)
																{
																	((DbsUsintTs_typ*)pFubInstance)->SetValue = TRUE;

																	((DbsUsintTs_typ*)pFubInstance)->FubRef.dbsUnit = DbsUnit;
																	((DbsUsintTs_typ*)pFubInstance)->FubRef.dbsDevice = cDBS_DEFAULT_DEVICE;
																	((DbsUsintTs_typ*)pFubInstance)->FubRef.dbsType = DbsType;
																	((DbsUsintTs_typ*)pFubInstance)->FubRef.dbsPoint = DbsPoint;
																	((DbsUsintTs_typ*)pFubInstance)->FubRef.dbsItem = i;
																	((DbsUsintTs_typ*)pFubInstance)->FubRef.countItem = pTypeDesc[DbsType].countItem;
																	((DbsUsintTs_typ*)pFubInstance)->FubRef.pidBrServer = 1;
																	((DbsUsintTs_typ*)pFubInstance)->FubRef.this = pFubInstance;

																	pFubInstanceDesc[countFubInstance].dbsUnit = DbsUnit;
																	pFubInstanceDesc[countFubInstance].dbsType = DbsType;
																	pFubInstanceDesc[countFubInstance].dbsPoint = DbsPoint;
																	pFubInstanceDesc[countFubInstance].dbsItem = i;
																	pFubInstanceDesc[countFubInstance].pFubInstance = (unsigned char*)pFubInstance;
																	countFubInstance++;
																}
																else if (pTypeDesc[DbsType].pItemDesc[i].idTypeItem == cDBS_IDTYPE_UINT &&
																	pTypeDesc[DbsType].pItemDesc[i].tsItem == FALSE)
																{
																	((DbsUint_typ*)pFubInstance)->SetValue = TRUE;

																	((DbsUint_typ*)pFubInstance)->FubRef.dbsUnit = DbsUnit;
																	((DbsUint_typ*)pFubInstance)->FubRef.dbsDevice = cDBS_DEFAULT_DEVICE;
																	((DbsUint_typ*)pFubInstance)->FubRef.dbsType = DbsType;
																	((DbsUint_typ*)pFubInstance)->FubRef.dbsPoint = DbsPoint;
																	((DbsUint_typ*)pFubInstance)->FubRef.dbsItem = i;
																	((DbsUint_typ*)pFubInstance)->FubRef.countItem = pTypeDesc[DbsType].countItem;
																	((DbsUint_typ*)pFubInstance)->FubRef.pidBrServer = 1;
																	((DbsUint_typ*)pFubInstance)->FubRef.this = pFubInstance;

																	pFubInstanceDesc[countFubInstance].dbsUnit = DbsUnit;
																	pFubInstanceDesc[countFubInstance].dbsType = DbsType;
																	pFubInstanceDesc[countFubInstance].dbsPoint = DbsPoint;
																	pFubInstanceDesc[countFubInstance].dbsItem = i;
																	pFubInstanceDesc[countFubInstance].pFubInstance = (unsigned char*)pFubInstance;
																	countFubInstance++;
																}
																else if (pTypeDesc[DbsType].pItemDesc[i].idTypeItem == cDBS_IDTYPE_INT &&
																	pTypeDesc[DbsType].pItemDesc[i].tsItem == FALSE)
																{
																	((DbsInt_typ*)pFubInstance)->SetValue = TRUE;

																	((DbsInt_typ*)pFubInstance)->FubRef.dbsUnit = DbsUnit;
																	((DbsInt_typ*)pFubInstance)->FubRef.dbsDevice = cDBS_DEFAULT_DEVICE;
																	((DbsInt_typ*)pFubInstance)->FubRef.dbsType = DbsType;
																	((DbsInt_typ*)pFubInstance)->FubRef.dbsPoint = DbsPoint;
																	((DbsInt_typ*)pFubInstance)->FubRef.dbsItem = i;
																	((DbsInt_typ*)pFubInstance)->FubRef.countItem = pTypeDesc[DbsType].countItem;
																	((DbsInt_typ*)pFubInstance)->FubRef.pidBrServer = 1;
																	((DbsInt_typ*)pFubInstance)->FubRef.this = pFubInstance;

																	pFubInstanceDesc[countFubInstance].dbsUnit = DbsUnit;
																	pFubInstanceDesc[countFubInstance].dbsType = DbsType;
																	pFubInstanceDesc[countFubInstance].dbsPoint = DbsPoint;
																	pFubInstanceDesc[countFubInstance].dbsItem = i;
																	pFubInstanceDesc[countFubInstance].pFubInstance = (unsigned char*)pFubInstance;
																	countFubInstance++;
																}
																else if (pTypeDesc[DbsType].pItemDesc[i].idTypeItem == cDBS_IDTYPE_UDINT &&
																	pTypeDesc[DbsType].pItemDesc[i].tsItem == FALSE)
																{
																	((DbsUdint_typ*)pFubInstance)->SetValue = TRUE;

																	((DbsUdint_typ*)pFubInstance)->FubRef.dbsUnit = DbsUnit;
																	((DbsUdint_typ*)pFubInstance)->FubRef.dbsDevice = cDBS_DEFAULT_DEVICE;
																	((DbsUdint_typ*)pFubInstance)->FubRef.dbsType = DbsType;
																	((DbsUdint_typ*)pFubInstance)->FubRef.dbsPoint = DbsPoint;
																	((DbsUdint_typ*)pFubInstance)->FubRef.dbsItem = i;
																	((DbsUdint_typ*)pFubInstance)->FubRef.countItem = pTypeDesc[DbsType].countItem;
																	((DbsUdint_typ*)pFubInstance)->FubRef.pidBrServer = 1;
																	((DbsUdint_typ*)pFubInstance)->FubRef.this = pFubInstance;

																	pFubInstanceDesc[countFubInstance].dbsUnit = DbsUnit;
																	pFubInstanceDesc[countFubInstance].dbsType = DbsType;
																	pFubInstanceDesc[countFubInstance].dbsPoint = DbsPoint;
																	pFubInstanceDesc[countFubInstance].dbsItem = i;
																	pFubInstanceDesc[countFubInstance].pFubInstance = (unsigned char*)pFubInstance;
																	countFubInstance++;
																}
																else if (pTypeDesc[DbsType].pItemDesc[i].idTypeItem == cDBS_IDTYPE_DINT &&
																	pTypeDesc[DbsType].pItemDesc[i].tsItem == FALSE)
																{
																	((DbsDint_typ*)pFubInstance)->SetValue = TRUE;

																	((DbsDint_typ*)pFubInstance)->FubRef.dbsUnit = DbsUnit;
																	((DbsDint_typ*)pFubInstance)->FubRef.dbsDevice = cDBS_DEFAULT_DEVICE;
																	((DbsDint_typ*)pFubInstance)->FubRef.dbsType = DbsType;
																	((DbsDint_typ*)pFubInstance)->FubRef.dbsPoint = DbsPoint;
																	((DbsDint_typ*)pFubInstance)->FubRef.dbsItem = i;
																	((DbsDint_typ*)pFubInstance)->FubRef.countItem = pTypeDesc[DbsType].countItem;
																	((DbsDint_typ*)pFubInstance)->FubRef.pidBrServer = 1;
																	((DbsDint_typ*)pFubInstance)->FubRef.this = pFubInstance;

																	pFubInstanceDesc[countFubInstance].dbsUnit = DbsUnit;
																	pFubInstanceDesc[countFubInstance].dbsType = DbsType;
																	pFubInstanceDesc[countFubInstance].dbsPoint = DbsPoint;
																	pFubInstanceDesc[countFubInstance].dbsItem = i;
																	pFubInstanceDesc[countFubInstance].pFubInstance = (unsigned char*)pFubInstance;
																	countFubInstance++;
																}
																if (flagDbsExistPoints == FALSE) {
																	flagDbsExistPoints = TRUE;
																	countExistPoints++;
																}
															} /* (stateFubInstance == 0) */
															else {
																countNotExistItems++;
																if (flagDbsNotExistPoints == FALSE) {
																	flagDbsNotExistPoints = TRUE;
																	countNotExistPoints++;
																}
															}
														}
													} /* (i=0; i<pTypeDesc[DbsType].countItem; i++) */
												} /* (flagDbsFub == TRUE) */
												else {
													countExistPoints++;
												}
											} /* (flagDbsUnit == TRUE && flagDbsType == TRUE && flagDbsPoint == TRUE) */
											break;
									} /* (SectionType) */
								} /* (pParser < (unsigned char*)pDA_Data + SizeDA_Data) */

								/* ---------------- */
								/* nächster Zustand */
								/* ---------------- */
								ParserState = cCD_PARSER_STATE_COMPARE_DO_POINT;

							} /* (StateTMP_alloc == 0) */
							else {
								/* Fehler bei TMP_alloc */
								ParserState = cCD_PARSER_STATE_ERROR;
							}
						} /* (StateTMP_alloc == 0) */
						else {
							/* Fehler bei TMP_alloc */
							ParserState = cCD_PARSER_STATE_ERROR;
						}
					} /* (StateTMP_alloc == 0) */
					else {
						/* Fehler bei TMP_alloc */
						ParserState = cCD_PARSER_STATE_ERROR;
					}
					break;

				/* ================================================ */
				/* DFA-Zustand: Abgleich der Datenpunktdefinitionen */
				/* ================================================ */
				case cCD_PARSER_STATE_COMPARE_DO_POINT:
					iDatObjInfo.enable = TRUE;
					iDatObjInfo.pName = (unsigned long)"DpDesc";
					DatObjInfo(&iDatObjInfo);
					if (iDatObjInfo.status == 0) {
						/* Datenmodul-Alignment beachten */
						if (iDatObjInfo.len >= countDefinedPoint * sizeof(POINT_DESC) &&
							iDatObjInfo.len <  countDefinedPoint * sizeof(POINT_DESC) + sizeof(unsigned long))
						{
							DbsPointChanged = FALSE;
							pWorkPointDesc = (POINT_DESC*)iDatObjInfo.pDatObjMem;
							for (i=0; i<countDefinedPoint; i++) {
								if (&pWorkPointDesc[i] >= (POINT_DESC*)(iDatObjInfo.pDatObjMem + iDatObjInfo.len)) {
									break;
								}
								if (pPointDesc[i].dbsUnit	== pWorkPointDesc[i].dbsUnit &&
									pPointDesc[i].dbsType	== pWorkPointDesc[i].dbsType &&
									pPointDesc[i].dbsPoint	== pWorkPointDesc[i].dbsPoint
								) {
								}
								else {
									DbsPointChanged = TRUE;
									break;
								}
							}
						}
						else {
							DbsPointChanged = TRUE;
						}
						if (DbsPointChanged == TRUE) {
							ParserState = cCD_PARSER_STATE_DEL_DO_POINT;
						}
						else {
							ParserState = cCD_PARSER_STATE_ALLOC_ACCESS_DATA;
						}
					}
					else if (iDatObjInfo.status == doERR_MODULNOTFOUND) {
						DbsPointChanged = TRUE;
						ParserState = cCD_PARSER_STATE_CREATE_DO_POINT;
					}
					else if (iDatObjInfo.status != ERR_FUB_BUSY) {
						ParserState = cCD_PARSER_STATE_ERROR;
					}
					break;
```
